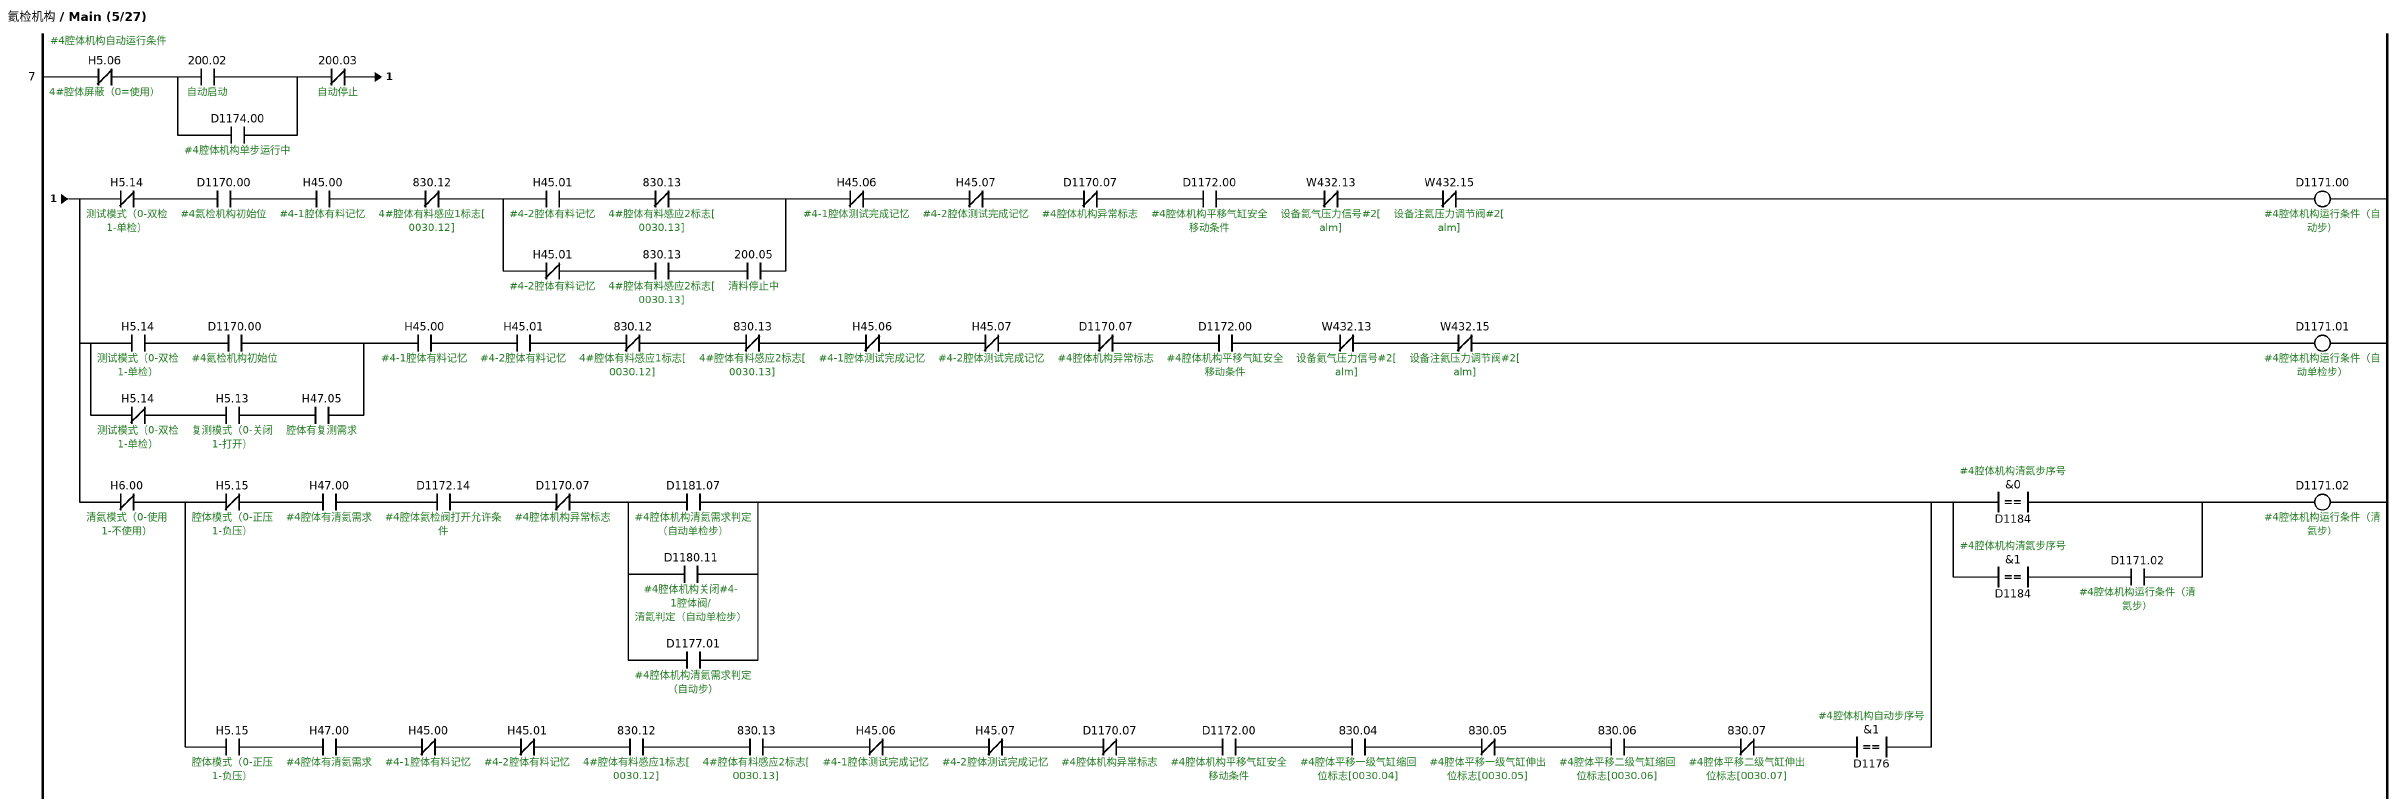
; [picture p144: 氦检机构 / Main, rungs 7-7]
; rung 7: #4腔体机构自动运行条件
LDNOT H5.06  ; 4#腔体屏蔽（0=使用）
LD 200.02  ; 自动启动
OR D1174.00  ; #4腔体机构单步运行中
ANDLD
ANDNOT 200.03  ; 自动停止
OUT TR0
ANDNOT H5.14  ; 测试模式（0-双检 1-单检）
AND D1170.00  ; #4氦检机构初始位
AND H45.00  ; #4-1腔体有料记忆
ANDNOT 830.12  ; 4#腔体有料感应1标志[0030.12]
LD H45.01  ; #4-2腔体有料记忆
ANDNOT 830.13  ; 4#腔体有料感应2标志[0030.13]
LDNOT H45.01  ; #4-2腔体有料记忆
AND 830.13  ; 4#腔体有料感应2标志[0030.13]
AND 200.05  ; 清料停止中
ORLD
ANDLD
ANDNOT H45.06  ; #4-1腔体测试完成记忆
ANDNOT H45.07  ; #4-2腔体测试完成记忆
ANDNOT D1170.07  ; #4腔体机构异常标志
AND D1172.00  ; #4腔体机构平移气缸安全移动条件
ANDNOT W432.13  ; 设备氦气压力信号#2[alm]
ANDNOT W432.15  ; 设备注氦压力调节阀#2[alm]
OUT D1171.00  ; #4腔体机构运行条件（自动步）
LD TR0
LD H5.14  ; 测试模式（0-双检 1-单检）
AND D1170.00  ; #4氦检机构初始位
LDNOT H5.14  ; 测试模式（0-双检 1-单检）
AND H5.13  ; 复测模式（0-关闭 1-打开）
AND H47.05  ; 腔体有复测需求
ORLD
ANDLD
AND H45.00  ; #4-1腔体有料记忆
AND H45.01  ; #4-2腔体有料记忆
ANDNOT 830.12  ; 4#腔体有料感应1标志[0030.12]
ANDNOT 830.13  ; 4#腔体有料感应2标志[0030.13]
ANDNOT H45.06  ; #4-1腔体测试完成记忆
ANDNOT H45.07  ; #4-2腔体测试完成记忆
ANDNOT D1170.07  ; #4腔体机构异常标志
AND D1172.00  ; #4腔体机构平移气缸安全移动条件
ANDNOT W432.13  ; 设备氦气压力信号#2[alm]
ANDNOT W432.15  ; 设备注氦压力调节阀#2[alm]
OUT D1171.01  ; #4腔体机构运行条件（自动单检步）
LD TR0
ANDNOT H6.00  ; 清氦模式（0-使用 1-不使用）
LDNOT H5.15  ; 腔体模式（0-正压 1-负压）
AND H47.00  ; #4腔体有清氦需求
AND D1172.14  ; #4腔体氦检阀打开允许条件
ANDNOT D1170.07  ; #4腔体机构异常标志
LD D1181.07  ; #4腔体机构清氦需求判定（自动单检步）
OR D1180.11  ; #4腔体机构关闭#4-1腔体阀/清氦判定（自动单检步）
OR D1177.01  ; #4腔体机构清氦需求判定（自动步）
ANDLD
LD H5.15  ; 腔体模式（0-正压 1-负压）
AND H47.00  ; #4腔体有清氦需求
ANDNOT H45.00  ; #4-1腔体有料记忆
ANDNOT H45.01  ; #4-2腔体有料记忆
AND 830.12  ; 4#腔体有料感应1标志[0030.12]
AND 830.13  ; 4#腔体有料感应2标志[0030.13]
ANDNOT H45.06  ; #4-1腔体测试完成记忆
ANDNOT H45.07  ; #4-2腔体测试完成记忆
ANDNOT D1170.07  ; #4腔体机构异常标志
AND D1172.00  ; #4腔体机构平移气缸安全移动条件
AND 830.04  ; #4腔体平移一级气缸缩回位标志[0030.04]
ANDNOT 830.05  ; #4腔体平移一级气缸伸出位标志[0030.05]
AND 830.06  ; #4腔体平移二级气缸缩回位标志[0030.06]
ANDNOT 830.07  ; #4腔体平移二级气缸伸出位标志[0030.07]
AND=L(301) &1 D1176  ; #4腔体机构自动步序号
ORLD
ANDLD
LD=L(301) &0 D1184  ; #4腔体机构清氦步序号
LD=L(301) &1 D1184  ; #4腔体机构清氦步序号
AND D1171.02  ; #4腔体机构运行条件（清氦步）
ORLD
ANDLD
OUT D1171.02  ; #4腔体机构运行条件（清氦步）

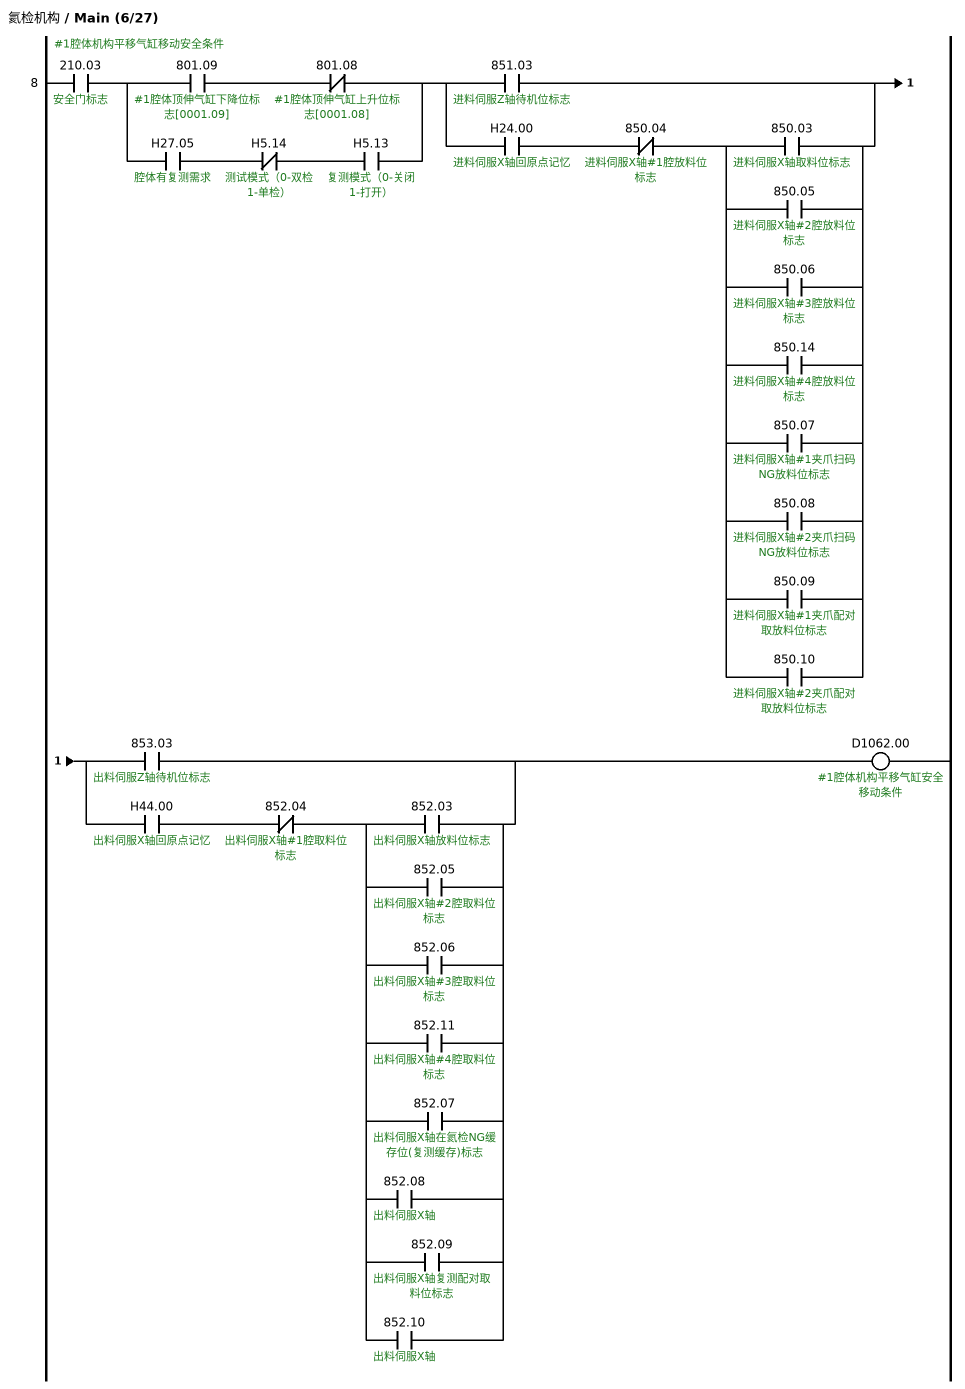
; rung 8: #1腔体机构平移气缸移动安全条件
LD 210.03  ; 安全门标志
LD 801.09  ; #1腔体顶伸气缸下降位标志[0001.09]
ANDNOT 801.08  ; #1腔体顶伸气缸上升位标志[0001.08]
LD H27.05  ; 腔体有复测需求
ANDNOT H5.14  ; 测试模式（0-双检 1-单检）
AND H5.13  ; 复测模式（0-关闭 1-打开）
ORLD
ANDLD
LD 851.03  ; 进料伺服Z轴待机位标志
LD H24.00  ; 进料伺服X轴回原点记忆
ANDNOT 850.04  ; 进料伺服X轴#1腔放料位标志
LD 850.03  ; 进料伺服X轴取料位标志
OR 850.05  ; 进料伺服X轴#2腔放料位标志
OR 850.06  ; 进料伺服X轴#3腔放料位标志
OR 850.14  ; 进料伺服X轴#4腔放料位标志
OR 850.07  ; 进料伺服X轴#1夹爪扫码NG放料位标志
OR 850.08  ; 进料伺服X轴#2夹爪扫码NG放料位标志
OR 850.09  ; 进料伺服X轴#1夹爪配对取放料位标志
OR 850.10  ; 进料伺服X轴#2夹爪配对取放料位标志
ANDLD
ORLD
ANDLD
LD 853.03  ; 出料伺服Z轴待机位标志
LD H44.00  ; 出料伺服X轴回原点记忆
ANDNOT 852.04  ; 出料伺服X轴#1腔取料位标志
LD 852.03  ; 出料伺服X轴放料位标志
OR 852.05  ; 出料伺服X轴#2腔取料位标志
OR 852.06  ; 出料伺服X轴#3腔取料位标志
OR 852.11  ; 出料伺服X轴#4腔取料位标志
OR 852.07  ; 出料伺服X轴在氦检NG缓存位(复测缓存)标志
OR 852.08  ; 出料伺服X轴
OR 852.09  ; 出料伺服X轴复测配对取料位标志
OR 852.10  ; 出料伺服X轴
ANDLD
ORLD
ANDLD
OUT D1062.00  ; #1腔体机构平移气缸安全移动条件

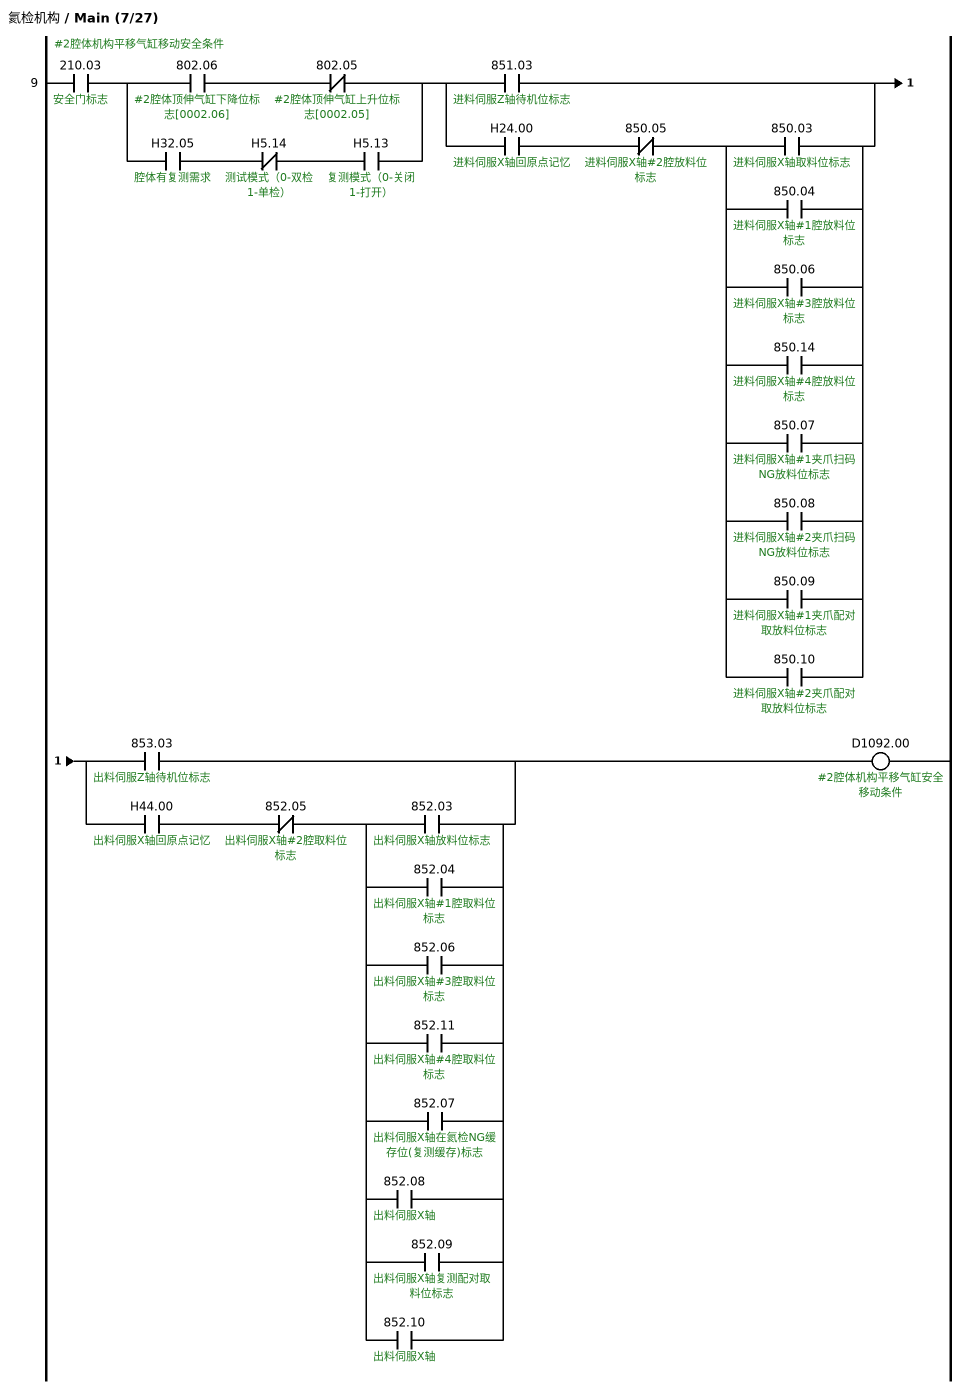
; rung 9: #2腔体机构平移气缸移动安全条件
LD 210.03  ; 安全门标志
LD 802.06  ; #2腔体顶伸气缸下降位标志[0002.06]
ANDNOT 802.05  ; #2腔体顶伸气缸上升位标志[0002.05]
LD H32.05  ; 腔体有复测需求
ANDNOT H5.14  ; 测试模式（0-双检 1-单检）
AND H5.13  ; 复测模式（0-关闭 1-打开）
ORLD
ANDLD
LD 851.03  ; 进料伺服Z轴待机位标志
LD H24.00  ; 进料伺服X轴回原点记忆
ANDNOT 850.05  ; 进料伺服X轴#2腔放料位标志
LD 850.03  ; 进料伺服X轴取料位标志
OR 850.04  ; 进料伺服X轴#1腔放料位标志
OR 850.06  ; 进料伺服X轴#3腔放料位标志
OR 850.14  ; 进料伺服X轴#4腔放料位标志
OR 850.07  ; 进料伺服X轴#1夹爪扫码NG放料位标志
OR 850.08  ; 进料伺服X轴#2夹爪扫码NG放料位标志
OR 850.09  ; 进料伺服X轴#1夹爪配对取放料位标志
OR 850.10  ; 进料伺服X轴#2夹爪配对取放料位标志
ANDLD
ORLD
ANDLD
LD 853.03  ; 出料伺服Z轴待机位标志
LD H44.00  ; 出料伺服X轴回原点记忆
ANDNOT 852.05  ; 出料伺服X轴#2腔取料位标志
LD 852.03  ; 出料伺服X轴放料位标志
OR 852.04  ; 出料伺服X轴#1腔取料位标志
OR 852.06  ; 出料伺服X轴#3腔取料位标志
OR 852.11  ; 出料伺服X轴#4腔取料位标志
OR 852.07  ; 出料伺服X轴在氦检NG缓存位(复测缓存)标志
OR 852.08  ; 出料伺服X轴
OR 852.09  ; 出料伺服X轴复测配对取料位标志
OR 852.10  ; 出料伺服X轴
ANDLD
ORLD
ANDLD
OUT D1092.00  ; #2腔体机构平移气缸安全移动条件

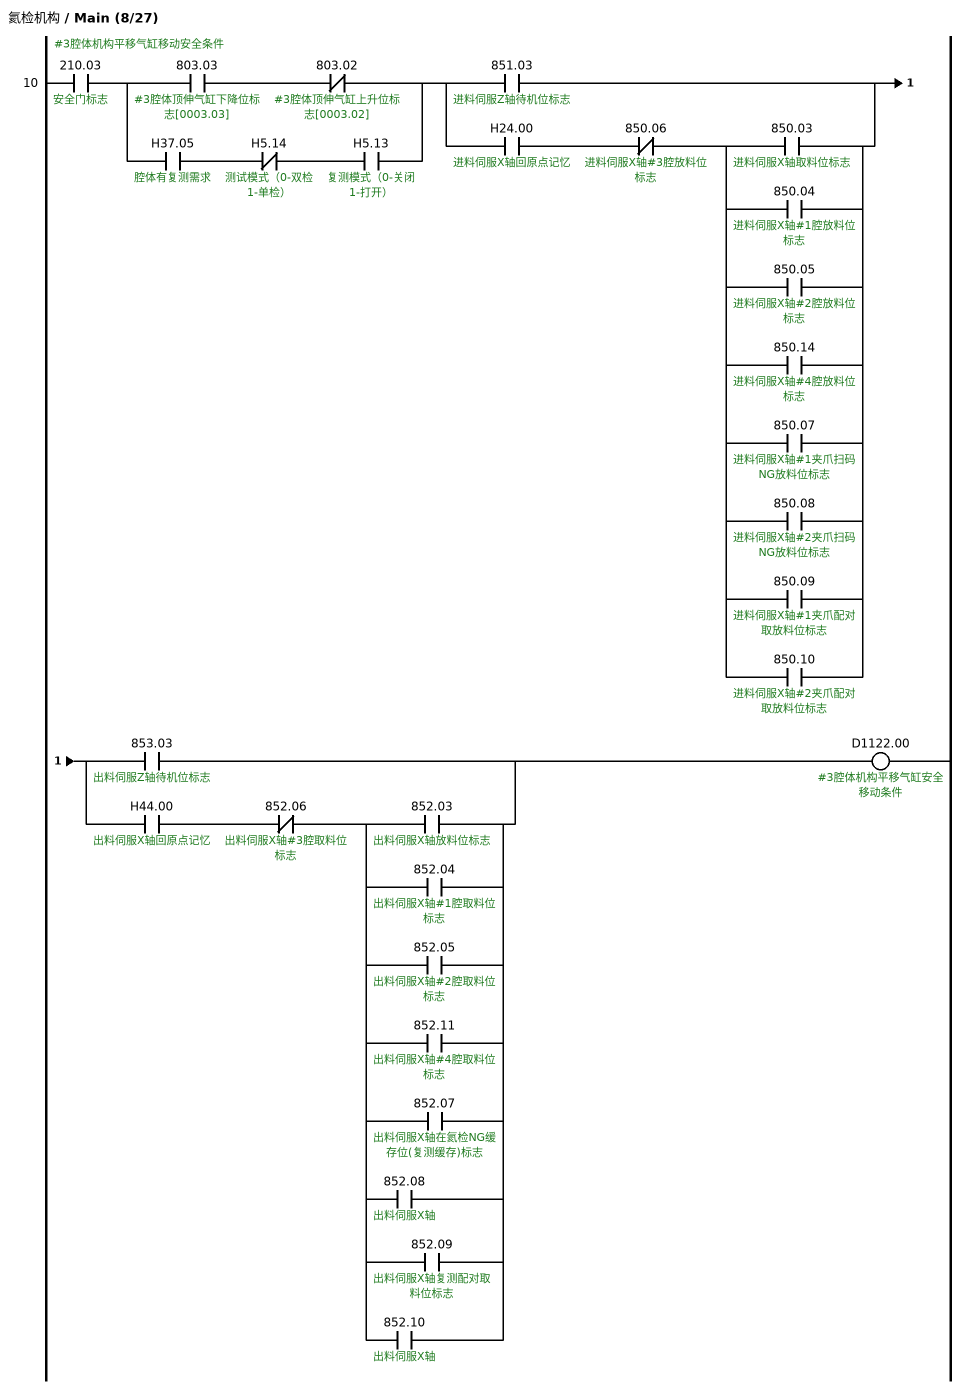
; rung 10: #3腔体机构平移气缸移动安全条件
LD 210.03  ; 安全门标志
LD 803.03  ; #3腔体顶伸气缸下降位标志[0003.03]
ANDNOT 803.02  ; #3腔体顶伸气缸上升位标志[0003.02]
LD H37.05  ; 腔体有复测需求
ANDNOT H5.14  ; 测试模式（0-双检 1-单检）
AND H5.13  ; 复测模式（0-关闭 1-打开）
ORLD
ANDLD
LD 851.03  ; 进料伺服Z轴待机位标志
LD H24.00  ; 进料伺服X轴回原点记忆
ANDNOT 850.06  ; 进料伺服X轴#3腔放料位标志
LD 850.03  ; 进料伺服X轴取料位标志
OR 850.04  ; 进料伺服X轴#1腔放料位标志
OR 850.05  ; 进料伺服X轴#2腔放料位标志
OR 850.14  ; 进料伺服X轴#4腔放料位标志
OR 850.07  ; 进料伺服X轴#1夹爪扫码NG放料位标志
OR 850.08  ; 进料伺服X轴#2夹爪扫码NG放料位标志
OR 850.09  ; 进料伺服X轴#1夹爪配对取放料位标志
OR 850.10  ; 进料伺服X轴#2夹爪配对取放料位标志
ANDLD
ORLD
ANDLD
LD 853.03  ; 出料伺服Z轴待机位标志
LD H44.00  ; 出料伺服X轴回原点记忆
ANDNOT 852.06  ; 出料伺服X轴#3腔取料位标志
LD 852.03  ; 出料伺服X轴放料位标志
OR 852.04  ; 出料伺服X轴#1腔取料位标志
OR 852.05  ; 出料伺服X轴#2腔取料位标志
OR 852.11  ; 出料伺服X轴#4腔取料位标志
OR 852.07  ; 出料伺服X轴在氦检NG缓存位(复测缓存)标志
OR 852.08  ; 出料伺服X轴
OR 852.09  ; 出料伺服X轴复测配对取料位标志
OR 852.10  ; 出料伺服X轴
ANDLD
ORLD
ANDLD
OUT D1122.00  ; #3腔体机构平移气缸安全移动条件

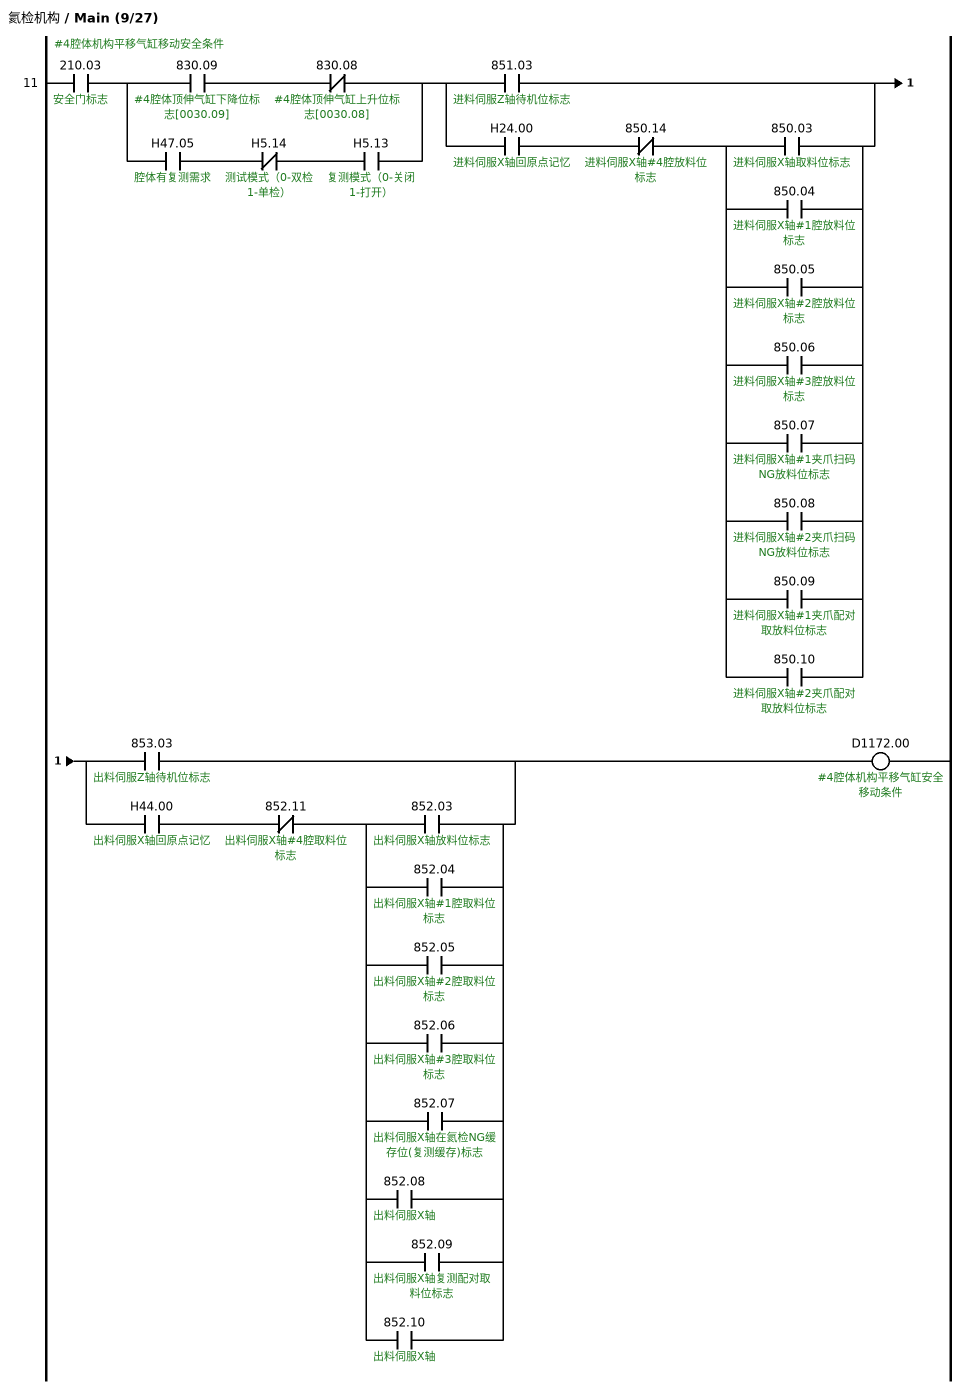
; rung 11: #4腔体机构平移气缸移动安全条件
LD 210.03  ; 安全门标志
LD 830.09  ; #4腔体顶伸气缸下降位标志[0030.09]
ANDNOT 830.08  ; #4腔体顶伸气缸上升位标志[0030.08]
LD H47.05  ; 腔体有复测需求
ANDNOT H5.14  ; 测试模式（0-双检 1-单检）
AND H5.13  ; 复测模式（0-关闭 1-打开）
ORLD
ANDLD
LD 851.03  ; 进料伺服Z轴待机位标志
LD H24.00  ; 进料伺服X轴回原点记忆
ANDNOT 850.14  ; 进料伺服X轴#4腔放料位标志
LD 850.03  ; 进料伺服X轴取料位标志
OR 850.04  ; 进料伺服X轴#1腔放料位标志
OR 850.05  ; 进料伺服X轴#2腔放料位标志
OR 850.06  ; 进料伺服X轴#3腔放料位标志
OR 850.07  ; 进料伺服X轴#1夹爪扫码NG放料位标志
OR 850.08  ; 进料伺服X轴#2夹爪扫码NG放料位标志
OR 850.09  ; 进料伺服X轴#1夹爪配对取放料位标志
OR 850.10  ; 进料伺服X轴#2夹爪配对取放料位标志
ANDLD
ORLD
ANDLD
LD 853.03  ; 出料伺服Z轴待机位标志
LD H44.00  ; 出料伺服X轴回原点记忆
ANDNOT 852.11  ; 出料伺服X轴#4腔取料位标志
LD 852.03  ; 出料伺服X轴放料位标志
OR 852.04  ; 出料伺服X轴#1腔取料位标志
OR 852.05  ; 出料伺服X轴#2腔取料位标志
OR 852.06  ; 出料伺服X轴#3腔取料位标志
OR 852.07  ; 出料伺服X轴在氦检NG缓存位(复测缓存)标志
OR 852.08  ; 出料伺服X轴
OR 852.09  ; 出料伺服X轴复测配对取料位标志
OR 852.10  ; 出料伺服X轴
ANDLD
ORLD
ANDLD
OUT D1172.00  ; #4腔体机构平移气缸安全移动条件

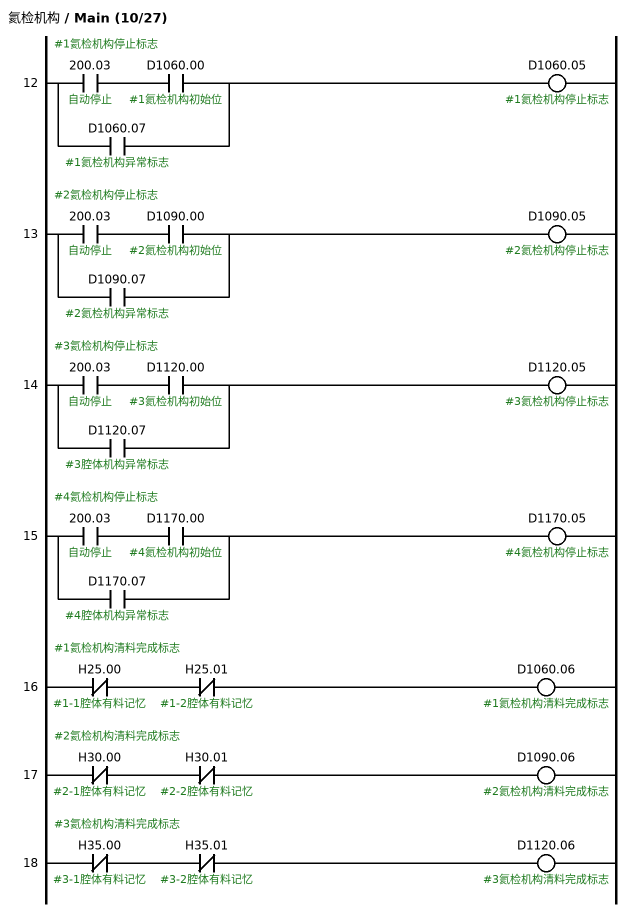
; rung 12: #1氦检机构停止标志
LD 200.03  ; 自动停止
AND D1060.00  ; #1氦检机构初始位
OR D1060.07  ; #1氦检机构异常标志
OUT D1060.05  ; #1氦检机构停止标志
; rung 13: #2氦检机构停止标志
LD 200.03  ; 自动停止
AND D1090.00  ; #2氦检机构初始位
OR D1090.07  ; #2氦检机构异常标志
OUT D1090.05  ; #2氦检机构停止标志
; rung 14: #3氦检机构停止标志
LD 200.03  ; 自动停止
AND D1120.00  ; #3氦检机构初始位
OR D1120.07  ; #3腔体机构异常标志
OUT D1120.05  ; #3氦检机构停止标志
; rung 15: #4氦检机构停止标志
LD 200.03  ; 自动停止
AND D1170.00  ; #4氦检机构初始位
OR D1170.07  ; #4腔体机构异常标志
OUT D1170.05  ; #4氦检机构停止标志
; rung 16: #1氦检机构清料完成标志
LDNOT H25.00  ; #1-1腔体有料记忆
ANDNOT H25.01  ; #1-2腔体有料记忆
OUT D1060.06  ; #1氦检机构清料完成标志
; rung 17: #2氦检机构清料完成标志
LDNOT H30.00  ; #2-1腔体有料记忆
ANDNOT H30.01  ; #2-2腔体有料记忆
OUT D1090.06  ; #2氦检机构清料完成标志
; rung 18: #3氦检机构清料完成标志
LDNOT H35.00  ; #3-1腔体有料记忆
ANDNOT H35.01  ; #3-2腔体有料记忆
OUT D1120.06  ; #3氦检机构清料完成标志

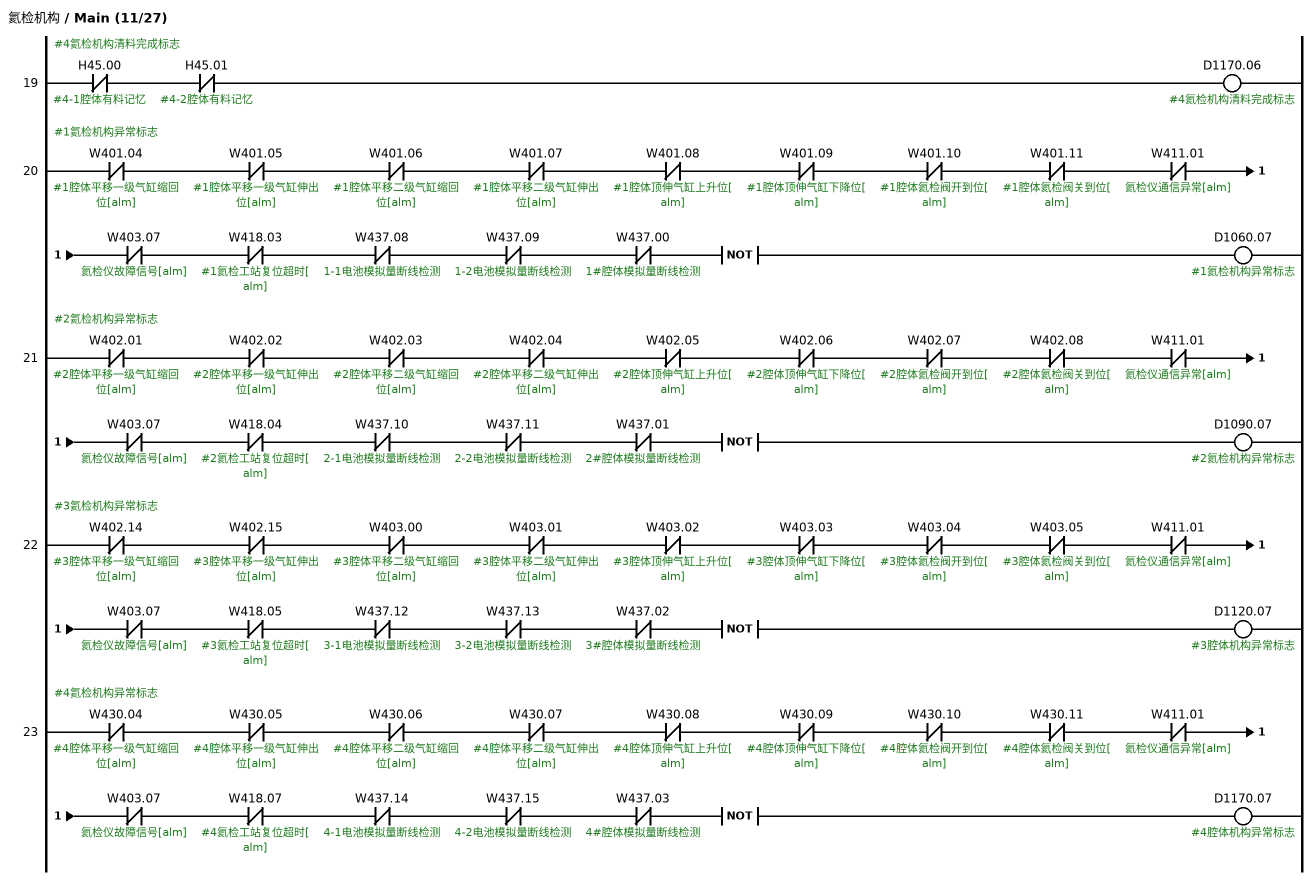
; rung 19: #4氦检机构清料完成标志
LDNOT H45.00  ; #4-1腔体有料记忆
ANDNOT H45.01  ; #4-2腔体有料记忆
OUT D1170.06  ; #4氦检机构清料完成标志
; rung 20: #1氦检机构异常标志
LDNOT W401.04  ; #1腔体平移一级气缸缩回位[alm]
ANDNOT W401.05  ; #1腔体平移一级气缸伸出位[alm]
ANDNOT W401.06  ; #1腔体平移二级气缸缩回位[alm]
ANDNOT W401.07  ; #1腔体平移二级气缸伸出位[alm]
ANDNOT W401.08  ; #1腔体顶伸气缸上升位[alm]
ANDNOT W401.09  ; #1腔体顶伸气缸下降位[alm]
ANDNOT W401.10  ; #1腔体氦检阀开到位[alm]
ANDNOT W401.11  ; #1腔体氦检阀关到位[alm]
ANDNOT W411.01  ; 氦检仪通信异常[alm]
ANDNOT W403.07  ; 氦检仪故障信号[alm]
ANDNOT W418.03  ; #1氦检工站复位超时[alm]
ANDNOT W437.08  ; 1-1电池模拟量断线检测
ANDNOT W437.09  ; 1-2电池模拟量断线检测
ANDNOT W437.00  ; 1#腔体模拟量断线检测
NOT(520)
OUT D1060.07  ; #1氦检机构异常标志
; rung 21: #2氦检机构异常标志
LDNOT W402.01  ; #2腔体平移一级气缸缩回位[alm]
ANDNOT W402.02  ; #2腔体平移一级气缸伸出位[alm]
ANDNOT W402.03  ; #2腔体平移二级气缸缩回位[alm]
ANDNOT W402.04  ; #2腔体平移二级气缸伸出位[alm]
ANDNOT W402.05  ; #2腔体顶伸气缸上升位[alm]
ANDNOT W402.06  ; #2腔体顶伸气缸下降位[alm]
ANDNOT W402.07  ; #2腔体氦检阀开到位[alm]
ANDNOT W402.08  ; #2腔体氦检阀关到位[alm]
ANDNOT W411.01  ; 氦检仪通信异常[alm]
ANDNOT W403.07  ; 氦检仪故障信号[alm]
ANDNOT W418.04  ; #2氦检工站复位超时[alm]
ANDNOT W437.10  ; 2-1电池模拟量断线检测
ANDNOT W437.11  ; 2-2电池模拟量断线检测
ANDNOT W437.01  ; 2#腔体模拟量断线检测
NOT(520)
OUT D1090.07  ; #2氦检机构异常标志
; rung 22: #3氦检机构异常标志
LDNOT W402.14  ; #3腔体平移一级气缸缩回位[alm]
ANDNOT W402.15  ; #3腔体平移一级气缸伸出位[alm]
ANDNOT W403.00  ; #3腔体平移二级气缸缩回位[alm]
ANDNOT W403.01  ; #3腔体平移二级气缸伸出位[alm]
ANDNOT W403.02  ; #3腔体顶伸气缸上升位[alm]
ANDNOT W403.03  ; #3腔体顶伸气缸下降位[alm]
ANDNOT W403.04  ; #3腔体氦检阀开到位[alm]
ANDNOT W403.05  ; #3腔体氦检阀关到位[alm]
ANDNOT W411.01  ; 氦检仪通信异常[alm]
ANDNOT W403.07  ; 氦检仪故障信号[alm]
ANDNOT W418.05  ; #3氦检工站复位超时[alm]
ANDNOT W437.12  ; 3-1电池模拟量断线检测
ANDNOT W437.13  ; 3-2电池模拟量断线检测
ANDNOT W437.02  ; 3#腔体模拟量断线检测
NOT(520)
OUT D1120.07  ; #3腔体机构异常标志
; rung 23: #4氦检机构异常标志
LDNOT W430.04  ; #4腔体平移一级气缸缩回位[alm]
ANDNOT W430.05  ; #4腔体平移一级气缸伸出位[alm]
ANDNOT W430.06  ; #4腔体平移二级气缸缩回位[alm]
ANDNOT W430.07  ; #4腔体平移二级气缸伸出位[alm]
ANDNOT W430.08  ; #4腔体顶伸气缸上升位[alm]
ANDNOT W430.09  ; #4腔体顶伸气缸下降位[alm]
ANDNOT W430.10  ; #4腔体氦检阀开到位[alm]
ANDNOT W430.11  ; #4腔体氦检阀关到位[alm]
ANDNOT W411.01  ; 氦检仪通信异常[alm]
ANDNOT W403.07  ; 氦检仪故障信号[alm]
ANDNOT W418.07  ; #4氦检工站复位超时[alm]
ANDNOT W437.14  ; 4-1电池模拟量断线检测
ANDNOT W437.15  ; 4-2电池模拟量断线检测
ANDNOT W437.03  ; 4#腔体模拟量断线检测
NOT(520)
OUT D1170.07  ; #4腔体机构异常标志

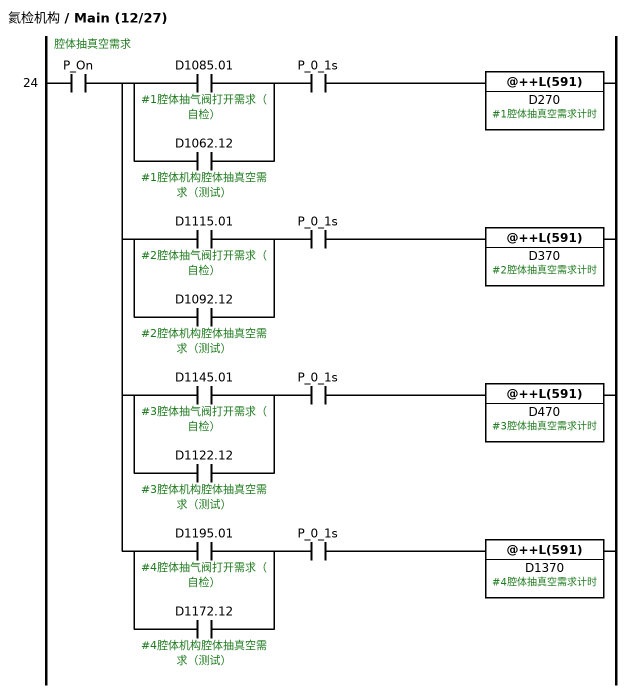
; rung 24: 腔体抽真空需求
LD P_On
OUT TR0
LD D1085.01  ; #1腔体抽气阀打开需求（自检）
OR D1062.12  ; #1腔体机构腔体抽真空需求（测试）
ANDLD
AND P_0_1s
@++L(591) D270  ; #1腔体抽真空需求计时
LD TR0
LD D1115.01  ; #2腔体抽气阀打开需求（自检）
OR D1092.12  ; #2腔体机构腔体抽真空需求（测试）
ANDLD
AND P_0_1s
@++L(591) D370  ; #2腔体抽真空需求计时
LD TR0
LD D1145.01  ; #3腔体抽气阀打开需求（自检）
OR D1122.12  ; #3腔体机构腔体抽真空需求（测试）
ANDLD
AND P_0_1s
@++L(591) D470  ; #3腔体抽真空需求计时
LD TR0
LD D1195.01  ; #4腔体抽气阀打开需求（自检）
OR D1172.12  ; #4腔体机构腔体抽真空需求（测试）
ANDLD
AND P_0_1s
@++L(591) D1370  ; #4腔体抽真空需求计时

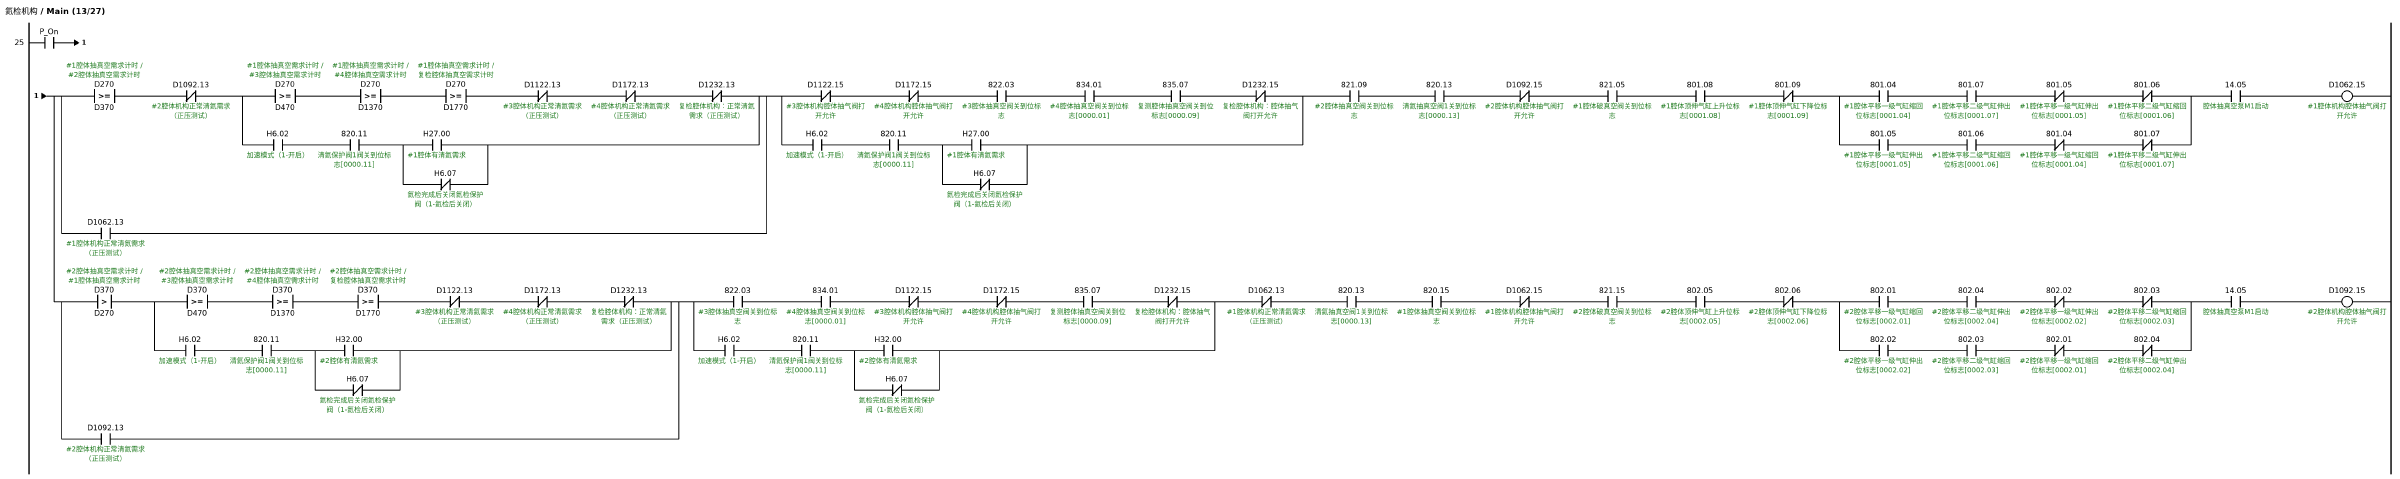
; rung 25
LD P_On
OUT TR0
LD>=L(326) D270 D370  ; #1腔体抽真空需求计时, #2腔体抽真空需求计时
ANDNOT D1092.13  ; #2腔体机构正常清氦需求（正压测试）
LD>=L(326) D270 D470  ; #1腔体抽真空需求计时, #3腔体抽真空需求计时
AND>=L(326) D270 D1370  ; #1腔体抽真空需求计时, #4腔体抽真空需求计时
AND>=L(326) D270 D1770  ; #1腔体抽真空需求计时, 复检腔体抽真空需求计时
ANDNOT D1122.13  ; #3腔体机构正常清氦需求（正压测试）
ANDNOT D1172.13  ; #4腔体机构正常清氦需求（正压测试）
ANDNOT D1232.13  ; 复检腔体机构：正常清氦需求（正压测试）
LD H6.02  ; 加速模式（1-开启）
AND 820.11  ; 清氦保护阀1阀关到位标志[0000.11]
LD H27.00  ; #1腔体有清氦需求
ORNOT H6.07  ; 氦检完成后关闭氦检保护阀（1-氦检后关闭）
ANDLD
ORLD
ANDLD
OR D1062.13  ; #1腔体机构正常清氦需求（正压测试）
ANDLD
LDNOT D1122.15  ; #3腔体机构腔体抽气阀打开允许
ANDNOT D1172.15  ; #4腔体机构腔体抽气阀打开允许
AND 822.03  ; #3腔体抽真空阀关到位标志
AND 834.01  ; #4腔体抽真空阀关到位标志[0000.01]
AND 835.07  ; 复测腔体抽真空阀关到位标志[0000.09]
ANDNOT D1232.15  ; 复检腔体机构：腔体抽气阀打开允许
LD H6.02  ; 加速模式（1-开启）
AND 820.11  ; 清氦保护阀1阀关到位标志[0000.11]
LD H27.00  ; #1腔体有清氦需求
ORNOT H6.07  ; 氦检完成后关闭氦检保护阀（1-氦检后关闭）
ANDLD
ORLD
ANDLD
AND 821.09  ; #2腔体抽真空阀关到位标志
AND 820.13  ; 清氦抽真空阀1关到位标志[0000.13]
ANDNOT D1092.15  ; #2腔体机构腔体抽气阀打开允许
AND 821.05  ; #1腔体破真空阀关到位标志
AND 801.08  ; #1腔体顶伸气缸上升位标志[0001.08]
ANDNOT 801.09  ; #1腔体顶伸气缸下降位标志[0001.09]
LD 801.04  ; #1腔体平移一级气缸缩回位标志[0001.04]
AND 801.07  ; #1腔体平移二级气缸伸出位标志[0001.07]
ANDNOT 801.05  ; #1腔体平移一级气缸伸出位标志[0001.05]
ANDNOT 801.06  ; #1腔体平移二级气缸缩回位标志[0001.06]
LD 801.05  ; #1腔体平移一级气缸伸出位标志[0001.05]
AND 801.06  ; #1腔体平移二级气缸缩回位标志[0001.06]
ANDNOT 801.04  ; #1腔体平移一级气缸缩回位标志[0001.04]
ANDNOT 801.07  ; #1腔体平移二级气缸伸出位标志[0001.07]
ORLD
ANDLD
AND 14.05  ; 腔体抽真空泵M1启动
OUT D1062.15  ; #1腔体机构腔体抽气阀打开允许
LD TR0
LD>L(321) D370 D270  ; #2腔体抽真空需求计时, #1腔体抽真空需求计时
LD>=L(326) D370 D470  ; #2腔体抽真空需求计时, #3腔体抽真空需求计时
AND>=L(326) D370 D1370  ; #2腔体抽真空需求计时, #4腔体抽真空需求计时
AND>=L(326) D370 D1770  ; #2腔体抽真空需求计时, 复检腔体抽真空需求计时
ANDNOT D1122.13  ; #3腔体机构正常清氦需求（正压测试）
ANDNOT D1172.13  ; #4腔体机构正常清氦需求（正压测试）
ANDNOT D1232.13  ; 复检腔体机构：正常清氦需求（正压测试）
LD H6.02  ; 加速模式（1-开启）
AND 820.11  ; 清氦保护阀1阀关到位标志[0000.11]
LD H32.00  ; #2腔体有清氦需求
ORNOT H6.07  ; 氦检完成后关闭氦检保护阀（1-氦检后关闭）
ANDLD
ORLD
ANDLD
OR D1092.13  ; #2腔体机构正常清氦需求（正压测试）
ANDLD
LD 822.03  ; #3腔体抽真空阀关到位标志
AND 834.01  ; #4腔体抽真空阀关到位标志[0000.01]
ANDNOT D1122.15  ; #3腔体机构腔体抽气阀打开允许
ANDNOT D1172.15  ; #4腔体机构腔体抽气阀打开允许
AND 835.07  ; 复测腔体抽真空阀关到位标志[0000.09]
ANDNOT D1232.15  ; 复检腔体机构：腔体抽气阀打开允许
LD H6.02  ; 加速模式（1-开启）
AND 820.11  ; 清氦保护阀1阀关到位标志[0000.11]
LD H32.00  ; #2腔体有清氦需求
ORNOT H6.07  ; 氦检完成后关闭氦检保护阀（1-氦检后关闭）
ANDLD
ORLD
ANDLD
ANDNOT D1062.13  ; #1腔体机构正常清氦需求（正压测试）
AND 820.13  ; 清氦抽真空阀1关到位标志[0000.13]
AND 820.15  ; #1腔体抽真空阀关到位标志
ANDNOT D1062.15  ; #1腔体机构腔体抽气阀打开允许
AND 821.15  ; #2腔体破真空阀关到位标志
AND 802.05  ; #2腔体顶伸气缸上升位标志[0002.05]
ANDNOT 802.06  ; #2腔体顶伸气缸下降位标志[0002.06]
LD 802.01  ; #2腔体平移一级气缸缩回位标志[0002.01]
AND 802.04  ; #2腔体平移二级气缸伸出位标志[0002.04]
ANDNOT 802.02  ; #2腔体平移一级气缸伸出位标志[0002.02]
ANDNOT 802.03  ; #2腔体平移二级气缸缩回位标志[0002.03]
LD 802.02  ; #2腔体平移一级气缸伸出位标志[0002.02]
AND 802.03  ; #2腔体平移二级气缸缩回位标志[0002.03]
ANDNOT 802.01  ; #2腔体平移一级气缸缩回位标志[0002.01]
ANDNOT 802.04  ; #2腔体平移二级气缸伸出位标志[0002.04]
ORLD
ANDLD
AND 14.05  ; 腔体抽真空泵M1启动
OUT D1092.15  ; #2腔体机构腔体抽气阀打开允许

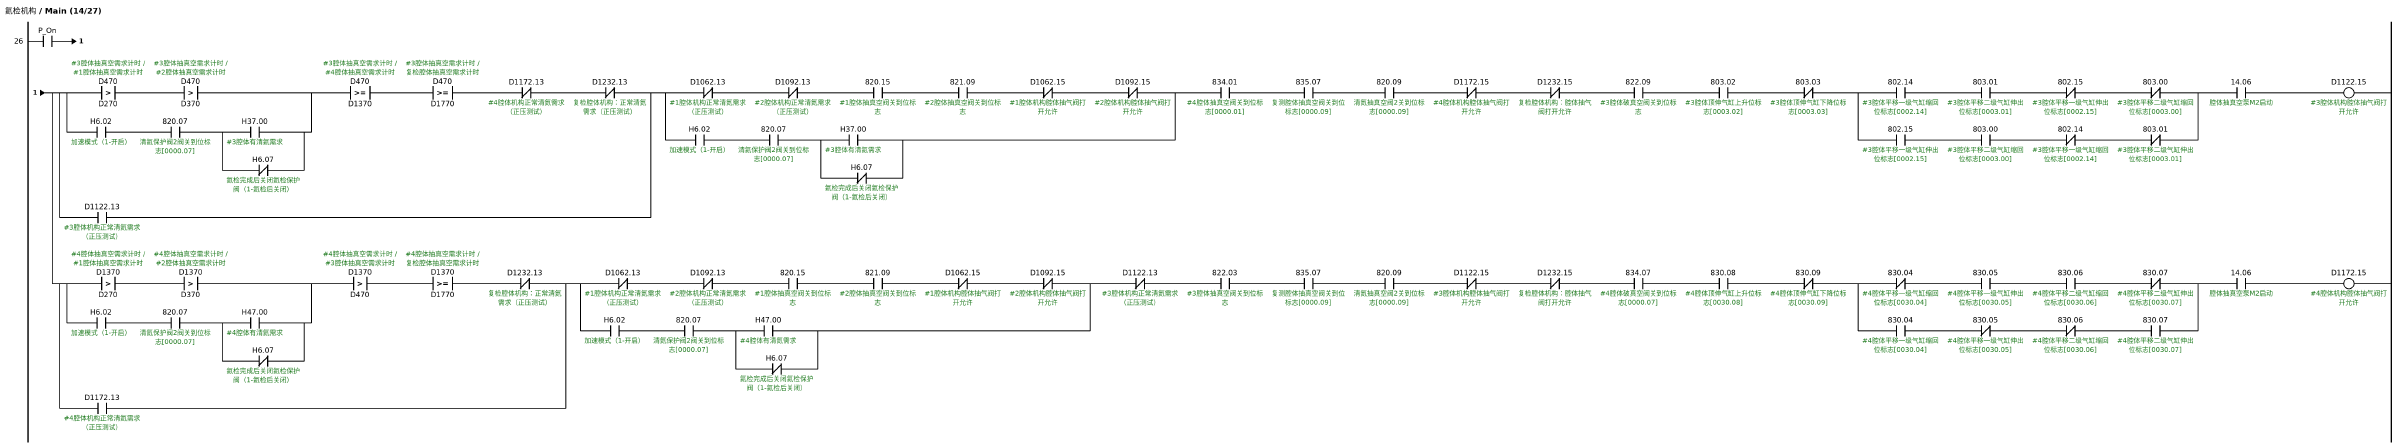
; rung 26
LD P_On
OUT TR0
LD>L(321) D470 D270  ; #3腔体抽真空需求计时, #1腔体抽真空需求计时
AND>L(321) D470 D370  ; #3腔体抽真空需求计时, #2腔体抽真空需求计时
LD H6.02  ; 加速模式（1-开启）
AND 820.07  ; 清氦保护阀2阀关到位标志[0000.07]
LD H37.00  ; #3腔体有清氦需求
ORNOT H6.07  ; 氦检完成后关闭氦检保护阀（1-氦检后关闭）
ANDLD
ORLD
AND>=L(326) D470 D1370  ; #3腔体抽真空需求计时, #4腔体抽真空需求计时
AND>=L(326) D470 D1770  ; #3腔体抽真空需求计时, 复检腔体抽真空需求计时
ANDNOT D1172.13  ; #4腔体机构正常清氦需求（正压测试）
ANDNOT D1232.13  ; 复检腔体机构：正常清氦需求（正压测试）
OR D1122.13  ; #3腔体机构正常清氦需求（正压测试）
ANDLD
LDNOT D1062.13  ; #1腔体机构正常清氦需求（正压测试）
ANDNOT D1092.13  ; #2腔体机构正常清氦需求（正压测试）
AND 820.15  ; #1腔体抽真空阀关到位标志
AND 821.09  ; #2腔体抽真空阀关到位标志
ANDNOT D1062.15  ; #1腔体机构腔体抽气阀打开允许
ANDNOT D1092.15  ; #2腔体机构腔体抽气阀打开允许
LD H6.02  ; 加速模式（1-开启）
AND 820.07  ; 清氦保护阀2阀关到位标志[0000.07]
LD H37.00  ; #3腔体有清氦需求
ORNOT H6.07  ; 氦检完成后关闭氦检保护阀（1-氦检后关闭）
ANDLD
ORLD
ANDLD
AND 834.01  ; #4腔体抽真空阀关到位标志[0000.01]
AND 835.07  ; 复测腔体抽真空阀关到位标志[0000.09]
AND 820.09  ; 清氦抽真空阀2关到位标志[0000.09]
ANDNOT D1172.15  ; #4腔体机构腔体抽气阀打开允许
ANDNOT D1232.15  ; 复检腔体机构：腔体抽气阀打开允许
AND 822.09  ; #3腔体破真空阀关到位标志
AND 803.02  ; #3腔体顶伸气缸上升位标志[0003.02]
ANDNOT 803.03  ; #3腔体顶伸气缸下降位标志[0003.03]
LD 802.14  ; #3腔体平移一级气缸缩回位标志[0002.14]
AND 803.01  ; #3腔体平移二级气缸伸出位标志[0003.01]
ANDNOT 802.15  ; #3腔体平移一级气缸伸出位标志[0002.15]
ANDNOT 803.00  ; #3腔体平移二级气缸缩回位标志[0003.00]
LD 802.15  ; #3腔体平移一级气缸伸出位标志[0002.15]
AND 803.00  ; #3腔体平移二级气缸缩回位标志[0003.00]
ANDNOT 802.14  ; #3腔体平移一级气缸缩回位标志[0002.14]
ANDNOT 803.01  ; #3腔体平移二级气缸伸出位标志[0003.01]
ORLD
ANDLD
AND 14.06  ; 腔体抽真空泵M2启动
OUT D1122.15  ; #3腔体机构腔体抽气阀打开允许
LD TR0
LD>L(321) D1370 D270  ; #4腔体抽真空需求计时, #1腔体抽真空需求计时
AND>L(321) D1370 D370  ; #4腔体抽真空需求计时, #2腔体抽真空需求计时
LD H6.02  ; 加速模式（1-开启）
AND 820.07  ; 清氦保护阀2阀关到位标志[0000.07]
LD H47.00  ; #4腔体有清氦需求
ORNOT H6.07  ; 氦检完成后关闭氦检保护阀（1-氦检后关闭）
ANDLD
ORLD
AND>L(321) D1370 D470  ; #4腔体抽真空需求计时, #3腔体抽真空需求计时
AND>=L(326) D1370 D1770  ; #4腔体抽真空需求计时, 复检腔体抽真空需求计时
ANDNOT D1232.13  ; 复检腔体机构：正常清氦需求（正压测试）
OR D1172.13  ; #4腔体机构正常清氦需求（正压测试）
ANDLD
LDNOT D1062.13  ; #1腔体机构正常清氦需求（正压测试）
ANDNOT D1092.13  ; #2腔体机构正常清氦需求（正压测试）
AND 820.15  ; #1腔体抽真空阀关到位标志
AND 821.09  ; #2腔体抽真空阀关到位标志
ANDNOT D1062.15  ; #1腔体机构腔体抽气阀打开允许
ANDNOT D1092.15  ; #2腔体机构腔体抽气阀打开允许
LD H6.02  ; 加速模式（1-开启）
AND 820.07  ; 清氦保护阀2阀关到位标志[0000.07]
LD H47.00  ; #4腔体有清氦需求
ORNOT H6.07  ; 氦检完成后关闭氦检保护阀（1-氦检后关闭）
ANDLD
ORLD
ANDLD
ANDNOT D1122.13  ; #3腔体机构正常清氦需求（正压测试）
AND 822.03  ; #3腔体抽真空阀关到位标志
AND 835.07  ; 复测腔体抽真空阀关到位标志[0000.09]
AND 820.09  ; 清氦抽真空阀2关到位标志[0000.09]
ANDNOT D1122.15  ; #3腔体机构腔体抽气阀打开允许
ANDNOT D1232.15  ; 复检腔体机构：腔体抽气阀打开允许
AND 834.07  ; #4腔体破真空阀关到位标志[0000.07]
AND 830.08  ; #4腔体顶伸气缸上升位标志[0030.08]
ANDNOT 830.09  ; #4腔体顶伸气缸下降位标志[0030.09]
LDNOT 830.04  ; #4腔体平移一级气缸缩回位标志[0030.04]
AND 830.05  ; #4腔体平移一级气缸伸出位标志[0030.05]
AND 830.06  ; #4腔体平移二级气缸缩回位标志[0030.06]
ANDNOT 830.07  ; #4腔体平移二级气缸伸出位标志[0030.07]
LD 830.04  ; #4腔体平移一级气缸缩回位标志[0030.04]
ANDNOT 830.05  ; #4腔体平移一级气缸伸出位标志[0030.05]
ANDNOT 830.06  ; #4腔体平移二级气缸缩回位标志[0030.06]
AND 830.07  ; #4腔体平移二级气缸伸出位标志[0030.07]
ORLD
ANDLD
AND 14.06  ; 腔体抽真空泵M2启动
OUT D1172.15  ; #4腔体机构腔体抽气阀打开允许

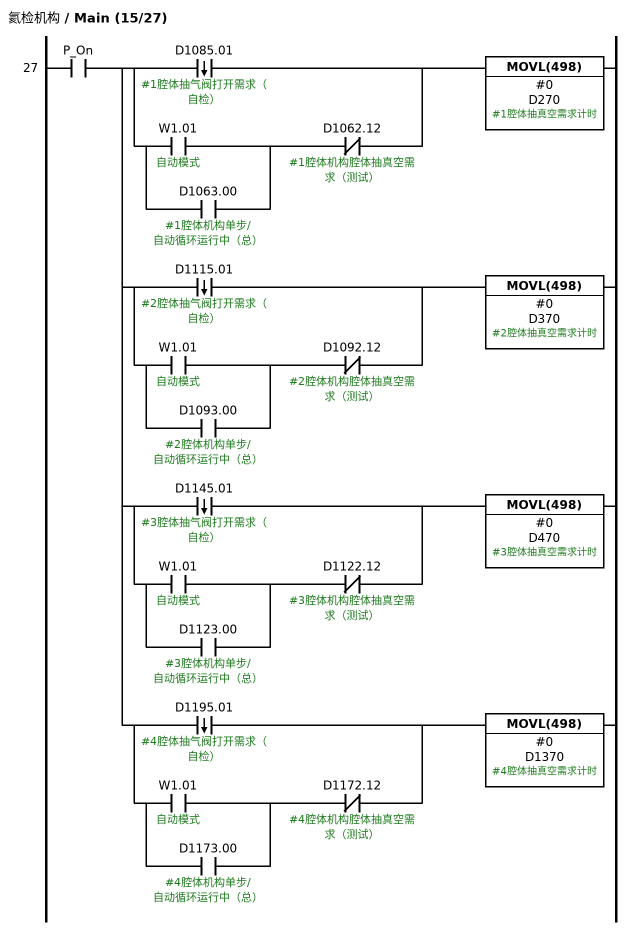
; rung 27
LD P_On
OUT TR0
%LD D1085.01  ; #1腔体抽气阀打开需求（自检）
LD W1.01  ; 自动模式
OR D1063.00  ; #1腔体机构单步/自动循环运行中（总）
ANDNOT D1062.12  ; #1腔体机构腔体抽真空需求（测试）
ORLD
ANDLD
MOVL(498) #0 D270  ; #1腔体抽真空需求计时
LD TR0
%LD D1115.01  ; #2腔体抽气阀打开需求（自检）
LD W1.01  ; 自动模式
OR D1093.00  ; #2腔体机构单步/自动循环运行中（总）
ANDNOT D1092.12  ; #2腔体机构腔体抽真空需求（测试）
ORLD
ANDLD
MOVL(498) #0 D370  ; #2腔体抽真空需求计时
LD TR0
%LD D1145.01  ; #3腔体抽气阀打开需求（自检）
LD W1.01  ; 自动模式
OR D1123.00  ; #3腔体机构单步/自动循环运行中（总）
ANDNOT D1122.12  ; #3腔体机构腔体抽真空需求（测试）
ORLD
ANDLD
MOVL(498) #0 D470  ; #3腔体抽真空需求计时
LD TR0
%LD D1195.01  ; #4腔体抽气阀打开需求（自检）
LD W1.01  ; 自动模式
OR D1173.00  ; #4腔体机构单步/自动循环运行中（总）
ANDNOT D1172.12  ; #4腔体机构腔体抽真空需求（测试）
ORLD
ANDLD
MOVL(498) #0 D1370  ; #4腔体抽真空需求计时

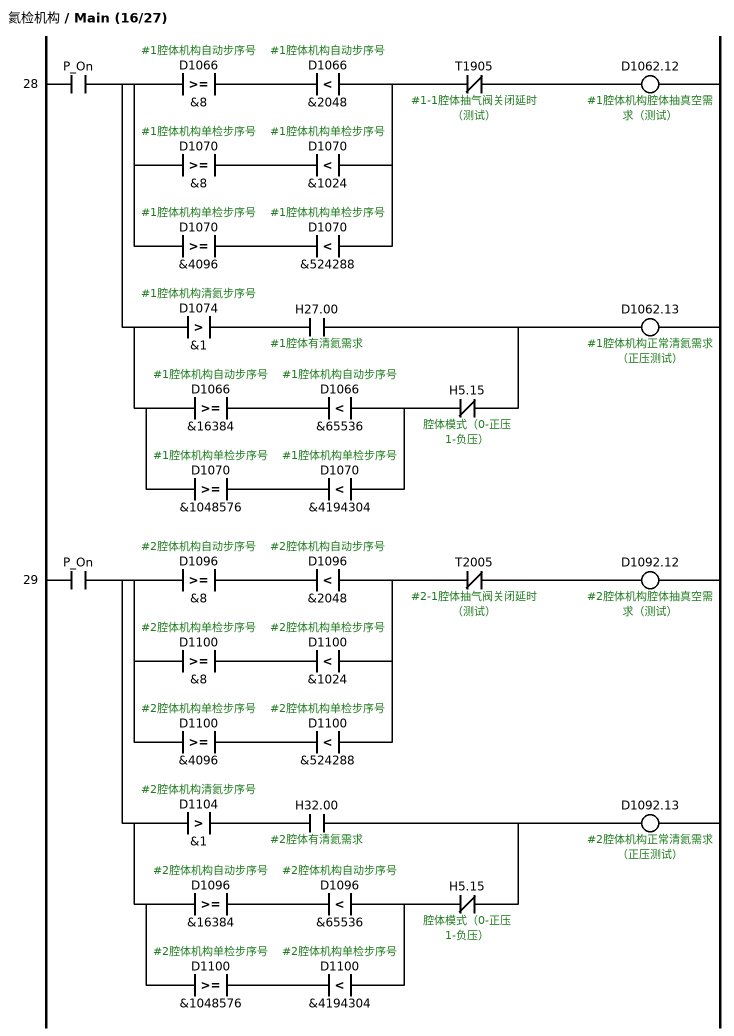
; rung 28
LD P_On
OUT TR0
LD>=L(326) D1066 &8  ; #1腔体机构自动步序号
AND<L(311) D1066 &2048  ; #1腔体机构自动步序号
LD>=L(326) D1070 &8  ; #1腔体机构单检步序号
AND<L(311) D1070 &1024  ; #1腔体机构单检步序号
ORLD
LD>=L(326) D1070 &4096  ; #1腔体机构单检步序号
AND<L(311) D1070 &524288  ; #1腔体机构单检步序号
ORLD
ANDLD
ANDNOT T1905  ; #1-1腔体抽气阀关闭延时（测试）
OUT D1062.12  ; #1腔体机构腔体抽真空需求（测试）
LD TR0
LD>L(321) D1074 &1  ; #1腔体机构清氦步序号
AND H27.00  ; #1腔体有清氦需求
LD>=L(326) D1066 &16384  ; #1腔体机构自动步序号
AND<L(311) D1066 &65536  ; #1腔体机构自动步序号
LD>=L(326) D1070 &1048576  ; #1腔体机构单检步序号
AND<L(311) D1070 &4194304  ; #1腔体机构单检步序号
ORLD
ANDNOT H5.15  ; 腔体模式（0-正压 1-负压）
ORLD
ANDLD
OUT D1062.13  ; #1腔体机构正常清氦需求（正压测试）
; rung 29
LD P_On
OUT TR0
LD>=L(326) D1096 &8  ; #2腔体机构自动步序号
AND<L(311) D1096 &2048  ; #2腔体机构自动步序号
LD>=L(326) D1100 &8  ; #2腔体机构单检步序号
AND<L(311) D1100 &1024  ; #2腔体机构单检步序号
ORLD
LD>=L(326) D1100 &4096  ; #2腔体机构单检步序号
AND<L(311) D1100 &524288  ; #2腔体机构单检步序号
ORLD
ANDLD
ANDNOT T2005  ; #2-1腔体抽气阀关闭延时（测试）
OUT D1092.12  ; #2腔体机构腔体抽真空需求（测试）
LD TR0
LD>L(321) D1104 &1  ; #2腔体机构清氦步序号
AND H32.00  ; #2腔体有清氦需求
LD>=L(326) D1096 &16384  ; #2腔体机构自动步序号
AND<L(311) D1096 &65536  ; #2腔体机构自动步序号
LD>=L(326) D1100 &1048576  ; #2腔体机构单检步序号
AND<L(311) D1100 &4194304  ; #2腔体机构单检步序号
ORLD
ANDNOT H5.15  ; 腔体模式（0-正压 1-负压）
ORLD
ANDLD
OUT D1092.13  ; #2腔体机构正常清氦需求（正压测试）

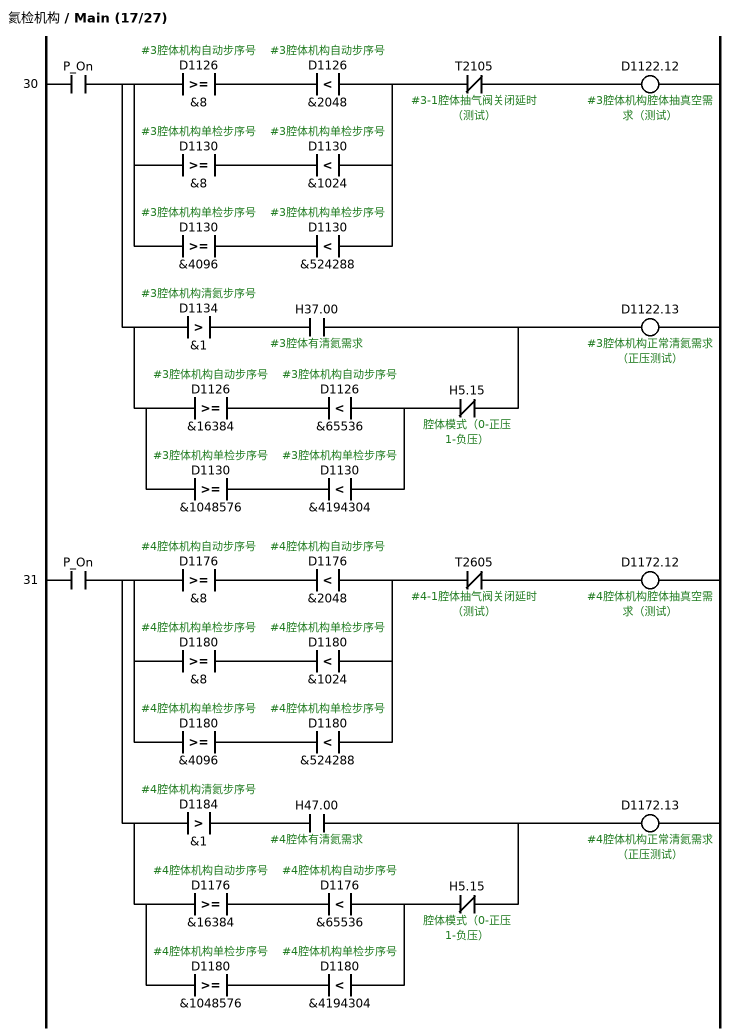
; rung 30
LD P_On
OUT TR0
LD>=L(326) D1126 &8  ; #3腔体机构自动步序号
AND<L(311) D1126 &2048  ; #3腔体机构自动步序号
LD>=L(326) D1130 &8  ; #3腔体机构单检步序号
AND<L(311) D1130 &1024  ; #3腔体机构单检步序号
ORLD
LD>=L(326) D1130 &4096  ; #3腔体机构单检步序号
AND<L(311) D1130 &524288  ; #3腔体机构单检步序号
ORLD
ANDLD
ANDNOT T2105  ; #3-1腔体抽气阀关闭延时（测试）
OUT D1122.12  ; #3腔体机构腔体抽真空需求（测试）
LD TR0
LD>L(321) D1134 &1  ; #3腔体机构清氦步序号
AND H37.00  ; #3腔体有清氦需求
LD>=L(326) D1126 &16384  ; #3腔体机构自动步序号
AND<L(311) D1126 &65536  ; #3腔体机构自动步序号
LD>=L(326) D1130 &1048576  ; #3腔体机构单检步序号
AND<L(311) D1130 &4194304  ; #3腔体机构单检步序号
ORLD
ANDNOT H5.15  ; 腔体模式（0-正压 1-负压）
ORLD
ANDLD
OUT D1122.13  ; #3腔体机构正常清氦需求（正压测试）
; rung 31
LD P_On
OUT TR0
LD>=L(326) D1176 &8  ; #4腔体机构自动步序号
AND<L(311) D1176 &2048  ; #4腔体机构自动步序号
LD>=L(326) D1180 &8  ; #4腔体机构单检步序号
AND<L(311) D1180 &1024  ; #4腔体机构单检步序号
ORLD
LD>=L(326) D1180 &4096  ; #4腔体机构单检步序号
AND<L(311) D1180 &524288  ; #4腔体机构单检步序号
ORLD
ANDLD
ANDNOT T2605  ; #4-1腔体抽气阀关闭延时（测试）
OUT D1172.12  ; #4腔体机构腔体抽真空需求（测试）
LD TR0
LD>L(321) D1184 &1  ; #4腔体机构清氦步序号
AND H47.00  ; #4腔体有清氦需求
LD>=L(326) D1176 &16384  ; #4腔体机构自动步序号
AND<L(311) D1176 &65536  ; #4腔体机构自动步序号
LD>=L(326) D1180 &1048576  ; #4腔体机构单检步序号
AND<L(311) D1180 &4194304  ; #4腔体机构单检步序号
ORLD
ANDNOT H5.15  ; 腔体模式（0-正压 1-负压）
ORLD
ANDLD
OUT D1172.13  ; #4腔体机构正常清氦需求（正压测试）

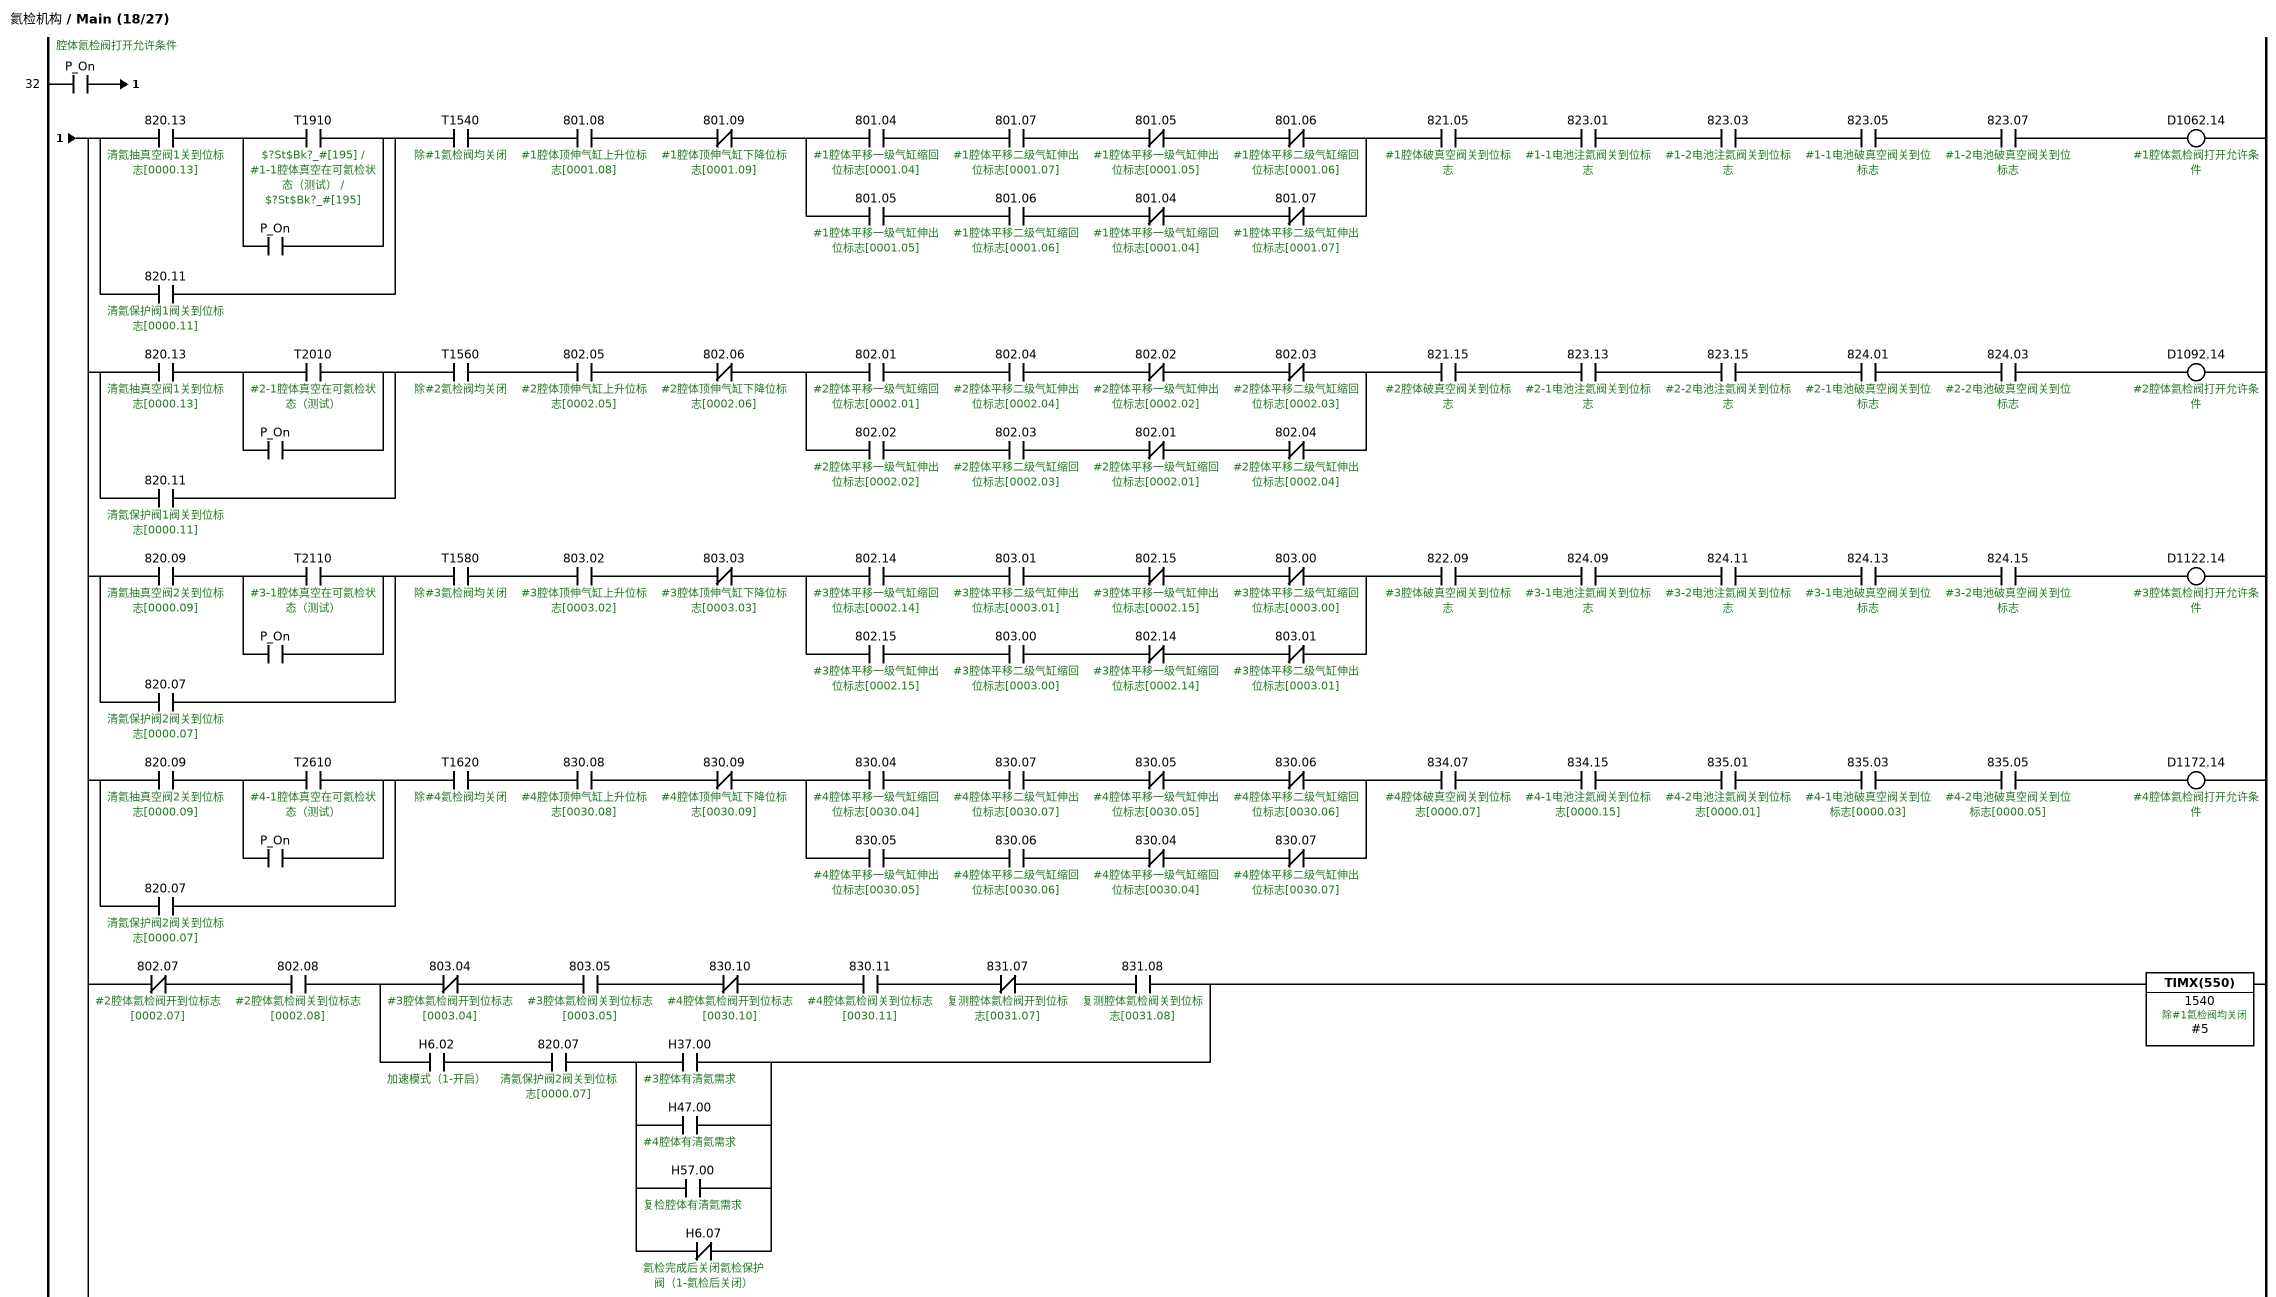

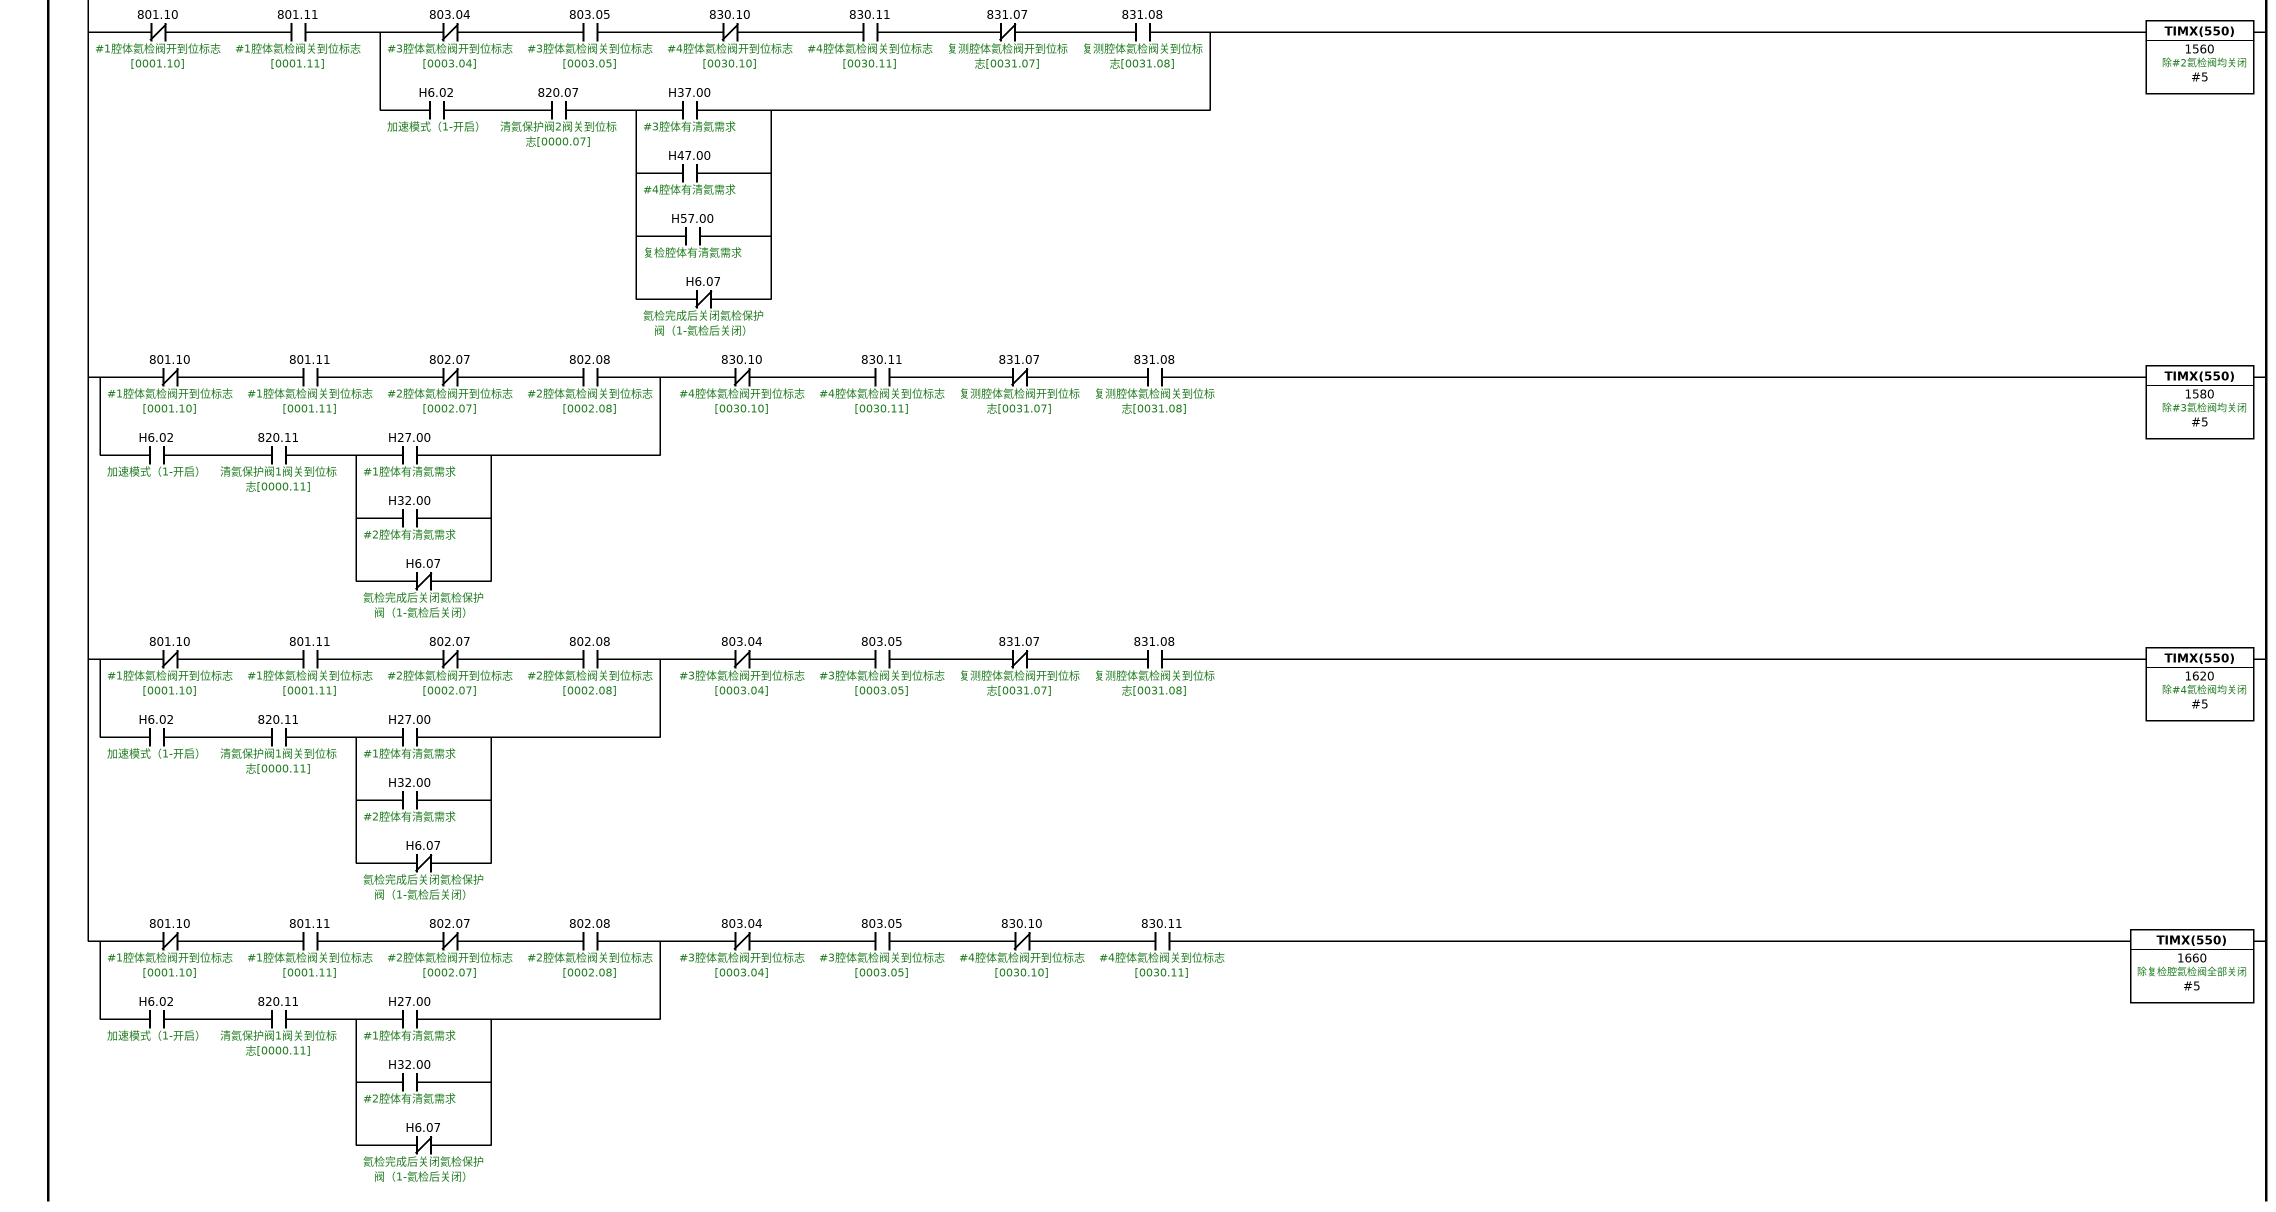
; rung 32: 腔体氦检阀打开允许条件
LD P_On
OUT TR0
LD 820.13  ; 清氦抽真空阀1关到位标志[0000.13]
LD T1910  ; $?St$Bk?_#[195] / #1-1腔体真空在可氦检状态（测试） / $?St$Bk?_#[195]
OR P_On
ANDLD
OR 820.11  ; 清氦保护阀1阀关到位标志[0000.11]
ANDLD
AND T1540  ; 除#1氦检阀均关闭
AND 801.08  ; #1腔体顶伸气缸上升位标志[0001.08]
ANDNOT 801.09  ; #1腔体顶伸气缸下降位标志[0001.09]
LD 801.04  ; #1腔体平移一级气缸缩回位标志[0001.04]
AND 801.07  ; #1腔体平移二级气缸伸出位标志[0001.07]
ANDNOT 801.05  ; #1腔体平移一级气缸伸出位标志[0001.05]
ANDNOT 801.06  ; #1腔体平移二级气缸缩回位标志[0001.06]
LD 801.05  ; #1腔体平移一级气缸伸出位标志[0001.05]
AND 801.06  ; #1腔体平移二级气缸缩回位标志[0001.06]
ANDNOT 801.04  ; #1腔体平移一级气缸缩回位标志[0001.04]
ANDNOT 801.07  ; #1腔体平移二级气缸伸出位标志[0001.07]
ORLD
ANDLD
AND 821.05  ; #1腔体破真空阀关到位标志
AND 823.01  ; #1-1电池注氦阀关到位标志
AND 823.03  ; #1-2电池注氦阀关到位标志
AND 823.05  ; #1-1电池破真空阀关到位标志
AND 823.07  ; #1-2电池破真空阀关到位标志
OUT D1062.14  ; #1腔体氦检阀打开允许条件
LD TR0
LD 820.13  ; 清氦抽真空阀1关到位标志[0000.13]
LD T2010  ; #2-1腔体真空在可氦检状态（测试）
OR P_On
ANDLD
OR 820.11  ; 清氦保护阀1阀关到位标志[0000.11]
ANDLD
AND T1560  ; 除#2氦检阀均关闭
AND 802.05  ; #2腔体顶伸气缸上升位标志[0002.05]
ANDNOT 802.06  ; #2腔体顶伸气缸下降位标志[0002.06]
LD 802.01  ; #2腔体平移一级气缸缩回位标志[0002.01]
AND 802.04  ; #2腔体平移二级气缸伸出位标志[0002.04]
ANDNOT 802.02  ; #2腔体平移一级气缸伸出位标志[0002.02]
ANDNOT 802.03  ; #2腔体平移二级气缸缩回位标志[0002.03]
LD 802.02  ; #2腔体平移一级气缸伸出位标志[0002.02]
AND 802.03  ; #2腔体平移二级气缸缩回位标志[0002.03]
ANDNOT 802.01  ; #2腔体平移一级气缸缩回位标志[0002.01]
ANDNOT 802.04  ; #2腔体平移二级气缸伸出位标志[0002.04]
ORLD
ANDLD
AND 821.15  ; #2腔体破真空阀关到位标志
AND 823.13  ; #2-1电池注氦阀关到位标志
AND 823.15  ; #2-2电池注氦阀关到位标志
AND 824.01  ; #2-1电池破真空阀关到位标志
AND 824.03  ; #2-2电池破真空阀关到位标志
OUT D1092.14  ; #2腔体氦检阀打开允许条件
LD TR0
LD 820.09  ; 清氦抽真空阀2关到位标志[0000.09]
LD T2110  ; #3-1腔体真空在可氦检状态（测试）
OR P_On
ANDLD
OR 820.07  ; 清氦保护阀2阀关到位标志[0000.07]
ANDLD
AND T1580  ; 除#3氦检阀均关闭
AND 803.02  ; #3腔体顶伸气缸上升位标志[0003.02]
ANDNOT 803.03  ; #3腔体顶伸气缸下降位标志[0003.03]
LD 802.14  ; #3腔体平移一级气缸缩回位标志[0002.14]
AND 803.01  ; #3腔体平移二级气缸伸出位标志[0003.01]
ANDNOT 802.15  ; #3腔体平移一级气缸伸出位标志[0002.15]
ANDNOT 803.00  ; #3腔体平移二级气缸缩回位标志[0003.00]
LD 802.15  ; #3腔体平移一级气缸伸出位标志[0002.15]
AND 803.00  ; #3腔体平移二级气缸缩回位标志[0003.00]
ANDNOT 802.14  ; #3腔体平移一级气缸缩回位标志[0002.14]
ANDNOT 803.01  ; #3腔体平移二级气缸伸出位标志[0003.01]
ORLD
ANDLD
AND 822.09  ; #3腔体破真空阀关到位标志
AND 824.09  ; #3-1电池注氦阀关到位标志
AND 824.11  ; #3-2电池注氦阀关到位标志
AND 824.13  ; #3-1电池破真空阀关到位标志
AND 824.15  ; #3-2电池破真空阀关到位标志
OUT D1122.14  ; #3腔体氦检阀打开允许条件
LD TR0
LD 820.09  ; 清氦抽真空阀2关到位标志[0000.09]
LD T2610  ; #4-1腔体真空在可氦检状态（测试）
OR P_On
ANDLD
OR 820.07  ; 清氦保护阀2阀关到位标志[0000.07]
ANDLD
AND T1620  ; 除#4氦检阀均关闭
AND 830.08  ; #4腔体顶伸气缸上升位标志[0030.08]
ANDNOT 830.09  ; #4腔体顶伸气缸下降位标志[0030.09]
LD 830.04  ; #4腔体平移一级气缸缩回位标志[0030.04]
AND 830.07  ; #4腔体平移二级气缸伸出位标志[0030.07]
ANDNOT 830.05  ; #4腔体平移一级气缸伸出位标志[0030.05]
ANDNOT 830.06  ; #4腔体平移二级气缸缩回位标志[0030.06]
LD 830.05  ; #4腔体平移一级气缸伸出位标志[0030.05]
AND 830.06  ; #4腔体平移二级气缸缩回位标志[0030.06]
ANDNOT 830.04  ; #4腔体平移一级气缸缩回位标志[0030.04]
ANDNOT 830.07  ; #4腔体平移二级气缸伸出位标志[0030.07]
ORLD
ANDLD
AND 834.07  ; #4腔体破真空阀关到位标志[0000.07]
AND 834.15  ; #4-1电池注氦阀关到位标志[0000.15]
AND 835.01  ; #4-2电池注氦阀关到位标志[0000.01]
AND 835.03  ; #4-1电池破真空阀关到位标志[0000.03]
AND 835.05  ; #4-2电池破真空阀关到位标志[0000.05]
OUT D1172.14  ; #4腔体氦检阀打开允许条件
LD TR0
ANDNOT 802.07  ; #2腔体氦检阀开到位标志[0002.07]
AND 802.08  ; #2腔体氦检阀关到位标志[0002.08]
LDNOT 803.04  ; #3腔体氦检阀开到位标志[0003.04]
AND 803.05  ; #3腔体氦检阀关到位标志[0003.05]
ANDNOT 830.10  ; #4腔体氦检阀开到位标志[0030.10]
AND 830.11  ; #4腔体氦检阀关到位标志[0030.11]
ANDNOT 831.07  ; 复测腔体氦检阀开到位标志[0031.07]
AND 831.08  ; 复测腔体氦检阀关到位标志[0031.08]
LD H6.02  ; 加速模式（1-开启）
AND 820.07  ; 清氦保护阀2阀关到位标志[0000.07]
LD H37.00  ; #3腔体有清氦需求
OR H47.00  ; #4腔体有清氦需求
OR H57.00  ; 复检腔体有清氦需求
ORNOT H6.07  ; 氦检完成后关闭氦检保护阀（1-氦检后关闭）
ANDLD
ORLD
ANDLD
TIMX(550) 1540 #5  ; 除#1氦检阀均关闭
LD TR0
ANDNOT 801.10  ; #1腔体氦检阀开到位标志[0001.10]
AND 801.11  ; #1腔体氦检阀关到位标志[0001.11]
LDNOT 803.04  ; #3腔体氦检阀开到位标志[0003.04]
AND 803.05  ; #3腔体氦检阀关到位标志[0003.05]
ANDNOT 830.10  ; #4腔体氦检阀开到位标志[0030.10]
AND 830.11  ; #4腔体氦检阀关到位标志[0030.11]
ANDNOT 831.07  ; 复测腔体氦检阀开到位标志[0031.07]
AND 831.08  ; 复测腔体氦检阀关到位标志[0031.08]
LD H6.02  ; 加速模式（1-开启）
AND 820.07  ; 清氦保护阀2阀关到位标志[0000.07]
LD H37.00  ; #3腔体有清氦需求
OR H47.00  ; #4腔体有清氦需求
OR H57.00  ; 复检腔体有清氦需求
ORNOT H6.07  ; 氦检完成后关闭氦检保护阀（1-氦检后关闭）
ANDLD
ORLD
ANDLD
TIMX(550) 1560 #5  ; 除#2氦检阀均关闭
LD TR0
LDNOT 801.10  ; #1腔体氦检阀开到位标志[0001.10]
AND 801.11  ; #1腔体氦检阀关到位标志[0001.11]
ANDNOT 802.07  ; #2腔体氦检阀开到位标志[0002.07]
AND 802.08  ; #2腔体氦检阀关到位标志[0002.08]
LD H6.02  ; 加速模式（1-开启）
AND 820.11  ; 清氦保护阀1阀关到位标志[0000.11]
LD H27.00  ; #1腔体有清氦需求
OR H32.00  ; #2腔体有清氦需求
ORNOT H6.07  ; 氦检完成后关闭氦检保护阀（1-氦检后关闭）
ANDLD
ORLD
ANDLD
ANDNOT 830.10  ; #4腔体氦检阀开到位标志[0030.10]
AND 830.11  ; #4腔体氦检阀关到位标志[0030.11]
ANDNOT 831.07  ; 复测腔体氦检阀开到位标志[0031.07]
AND 831.08  ; 复测腔体氦检阀关到位标志[0031.08]
TIMX(550) 1580 #5  ; 除#3氦检阀均关闭
LD TR0
LDNOT 801.10  ; #1腔体氦检阀开到位标志[0001.10]
AND 801.11  ; #1腔体氦检阀关到位标志[0001.11]
ANDNOT 802.07  ; #2腔体氦检阀开到位标志[0002.07]
AND 802.08  ; #2腔体氦检阀关到位标志[0002.08]
LD H6.02  ; 加速模式（1-开启）
AND 820.11  ; 清氦保护阀1阀关到位标志[0000.11]
LD H27.00  ; #1腔体有清氦需求
OR H32.00  ; #2腔体有清氦需求
ORNOT H6.07  ; 氦检完成后关闭氦检保护阀（1-氦检后关闭）
ANDLD
ORLD
ANDLD
ANDNOT 803.04  ; #3腔体氦检阀开到位标志[0003.04]
AND 803.05  ; #3腔体氦检阀关到位标志[0003.05]
ANDNOT 831.07  ; 复测腔体氦检阀开到位标志[0031.07]
AND 831.08  ; 复测腔体氦检阀关到位标志[0031.08]
TIMX(550) 1620 #5  ; 除#4氦检阀均关闭
LD TR0
LDNOT 801.10  ; #1腔体氦检阀开到位标志[0001.10]
AND 801.11  ; #1腔体氦检阀关到位标志[0001.11]
ANDNOT 802.07  ; #2腔体氦检阀开到位标志[0002.07]
AND 802.08  ; #2腔体氦检阀关到位标志[0002.08]
LD H6.02  ; 加速模式（1-开启）
AND 820.11  ; 清氦保护阀1阀关到位标志[0000.11]
LD H27.00  ; #1腔体有清氦需求
OR H32.00  ; #2腔体有清氦需求
ORNOT H6.07  ; 氦检完成后关闭氦检保护阀（1-氦检后关闭）
ANDLD
ORLD
ANDLD
ANDNOT 803.04  ; #3腔体氦检阀开到位标志[0003.04]
AND 803.05  ; #3腔体氦检阀关到位标志[0003.05]
ANDNOT 830.10  ; #4腔体氦检阀开到位标志[0030.10]
AND 830.11  ; #4腔体氦检阀关到位标志[0030.11]
TIMX(550) 1660 #5  ; 除复检腔氦检阀全部关闭

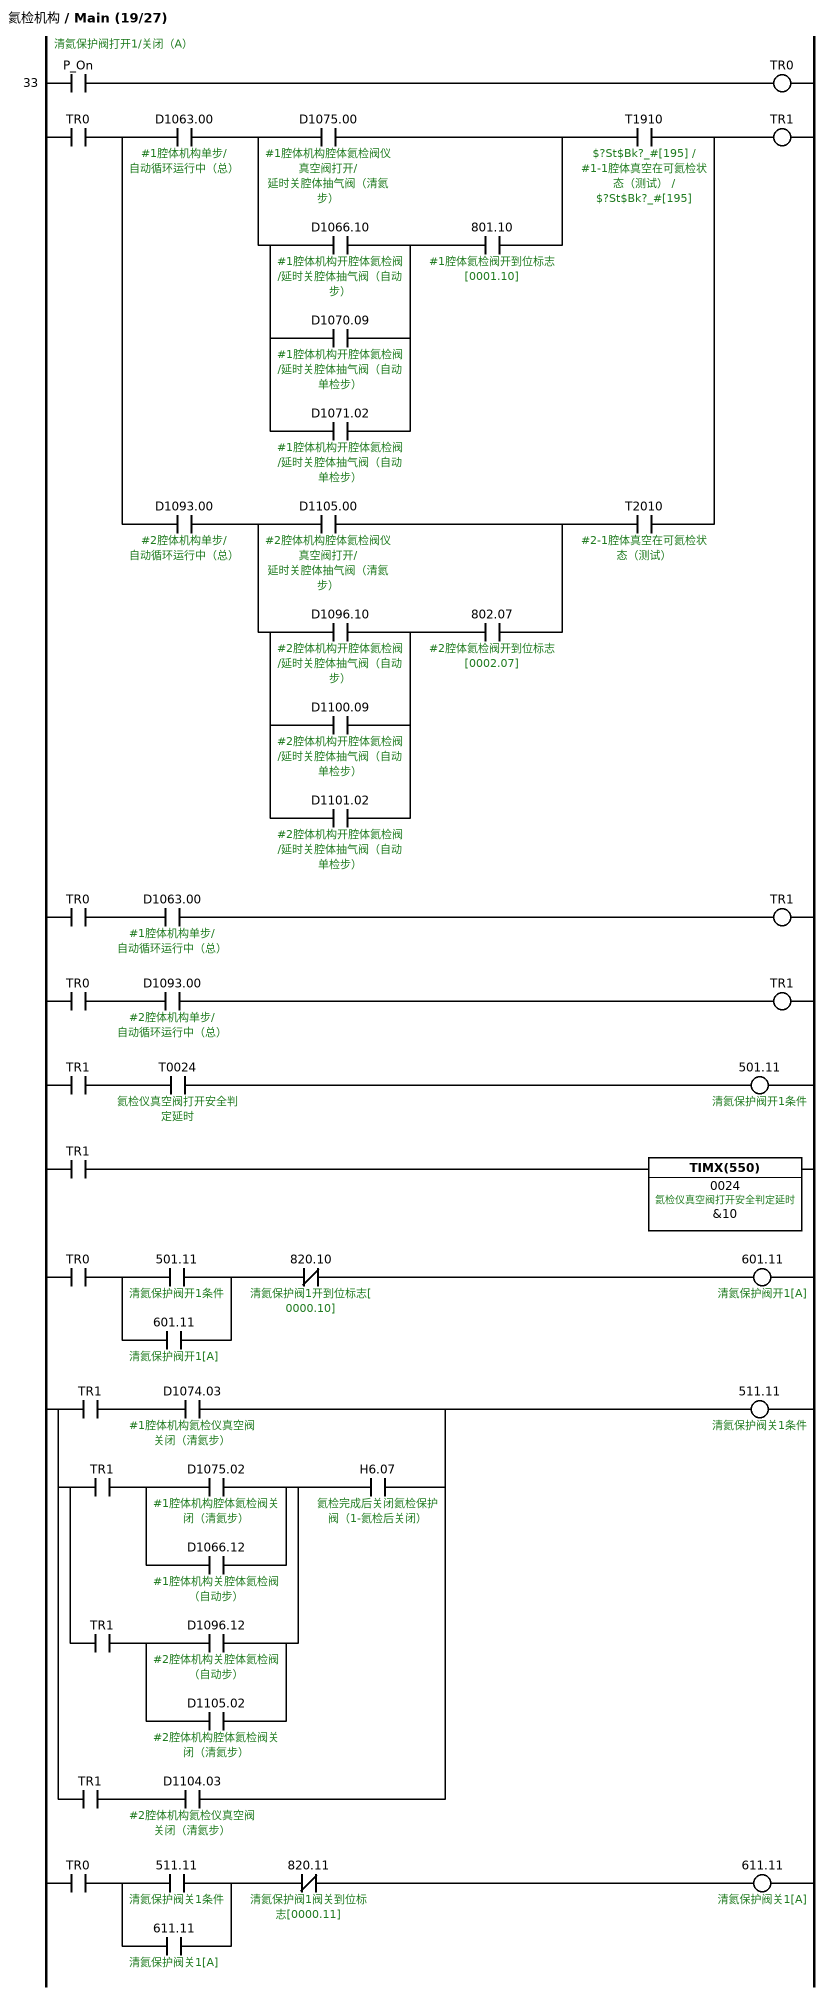
; rung 33: 清氦保护阀打开1/关闭（A）
LD P_On
OUT TR0
LD D1063.00  ; #1腔体机构单步/自动循环运行中（总）
LD D1075.00  ; #1腔体机构腔体氦检阀仪真空阀打开/延时关腔体抽气阀（清氦步）
LD D1066.10  ; #1腔体机构开腔体氦检阀/延时关腔体抽气阀（自动步）
OR D1070.09  ; #1腔体机构开腔体氦检阀/延时关腔体抽气阀（自动单检步）
OR D1071.02  ; #1腔体机构开腔体氦检阀/延时关腔体抽气阀（自动单检步）
AND 801.10  ; #1腔体氦检阀开到位标志[0001.10]
ORLD
ANDLD
AND T1910  ; $?St$Bk?_#[195] / #1-1腔体真空在可氦检状态（测试） / $?St$Bk?_#[195]
LD D1093.00  ; #2腔体机构单步/自动循环运行中（总）
LD D1105.00  ; #2腔体机构腔体氦检阀仪真空阀打开/延时关腔体抽气阀（清氦步）
LD D1096.10  ; #2腔体机构开腔体氦检阀/延时关腔体抽气阀（自动步）
OR D1100.09  ; #2腔体机构开腔体氦检阀/延时关腔体抽气阀（自动单检步）
OR D1101.02  ; #2腔体机构开腔体氦检阀/延时关腔体抽气阀（自动单检步）
AND 802.07  ; #2腔体氦检阀开到位标志[0002.07]
ORLD
ANDLD
AND T2010  ; #2-1腔体真空在可氦检状态（测试）
ORLD
ANDLD
OUT TR1
AND T0024  ; 氦检仪真空阀打开安全判定延时
OUT 501.11  ; 清氦保护阀开1条件
LD TR1
TIMX(550) 0024 &10  ; 氦检仪真空阀打开安全判定延时
LD TR0
LD 501.11  ; 清氦保护阀开1条件
OR 601.11  ; 清氦保护阀开1[A]
ANDLD
ANDNOT 820.10  ; 清氦保护阀1开到位标志[0000.10]
OUT 601.11  ; 清氦保护阀开1[A]
LD TR0
AND D1063.00  ; #1腔体机构单步/自动循环运行中（总）
OUT TR1
AND D1074.03  ; #1腔体机构氦检仪真空阀关闭（清氦步）
LD TR1
LD D1075.02  ; #1腔体机构腔体氦检阀关闭（清氦步）
OR D1066.12  ; #1腔体机构关腔体氦检阀（自动步）
ANDLD
LD TR0
AND D1093.00  ; #2腔体机构单步/自动循环运行中（总）
OUT TR1
LD D1096.12  ; #2腔体机构关腔体氦检阀（自动步）
OR D1105.02  ; #2腔体机构腔体氦检阀关闭（清氦步）
ANDLD
ORLD
AND H6.07  ; 氦检完成后关闭氦检保护阀（1-氦检后关闭）
ORLD
LD TR1
AND D1104.03  ; #2腔体机构氦检仪真空阀关闭（清氦步）
ORLD
OUT 511.11  ; 清氦保护阀关1条件
LD TR0
LD 511.11  ; 清氦保护阀关1条件
OR 611.11  ; 清氦保护阀关1[A]
ANDLD
ANDNOT 820.11  ; 清氦保护阀1阀关到位标志[0000.11]
OUT 611.11  ; 清氦保护阀关1[A]

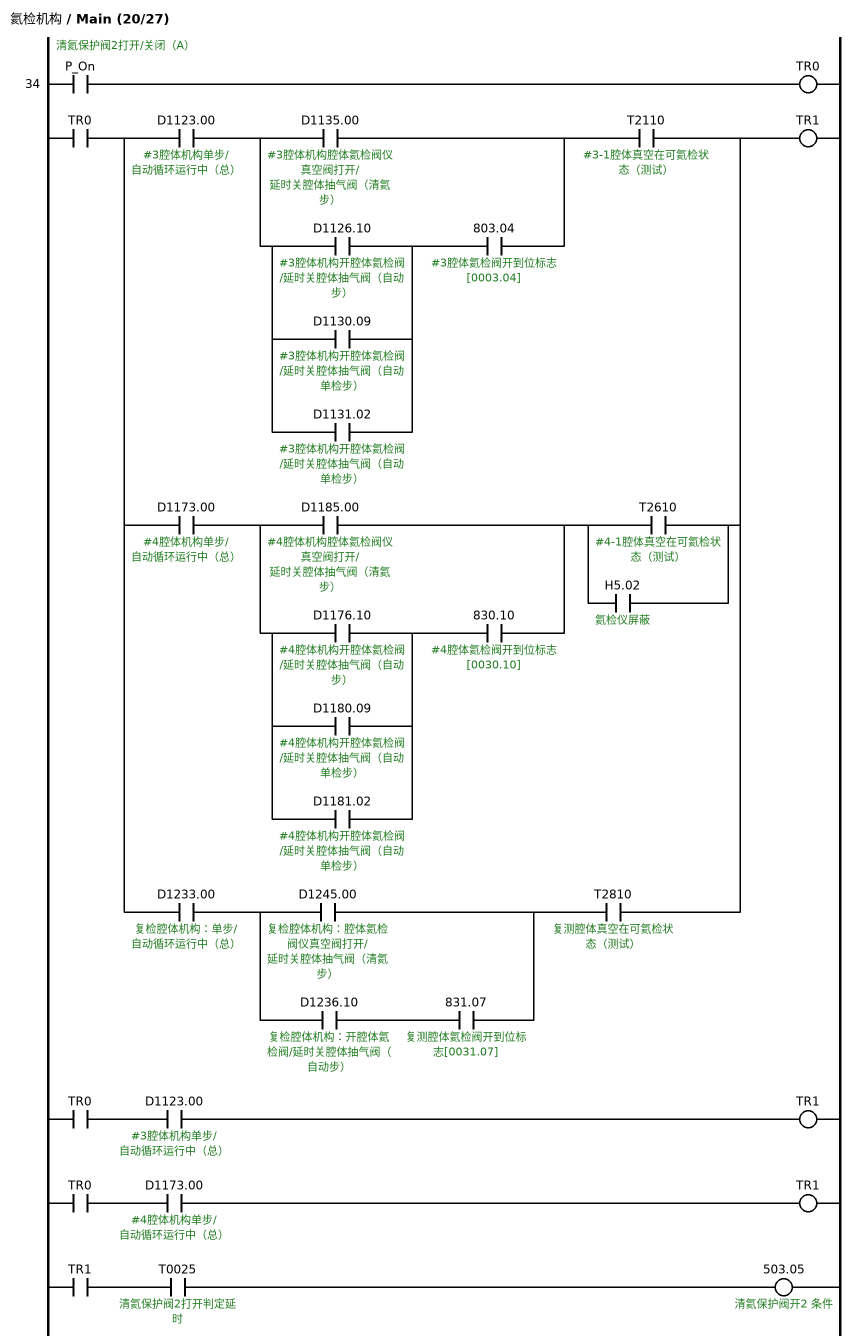

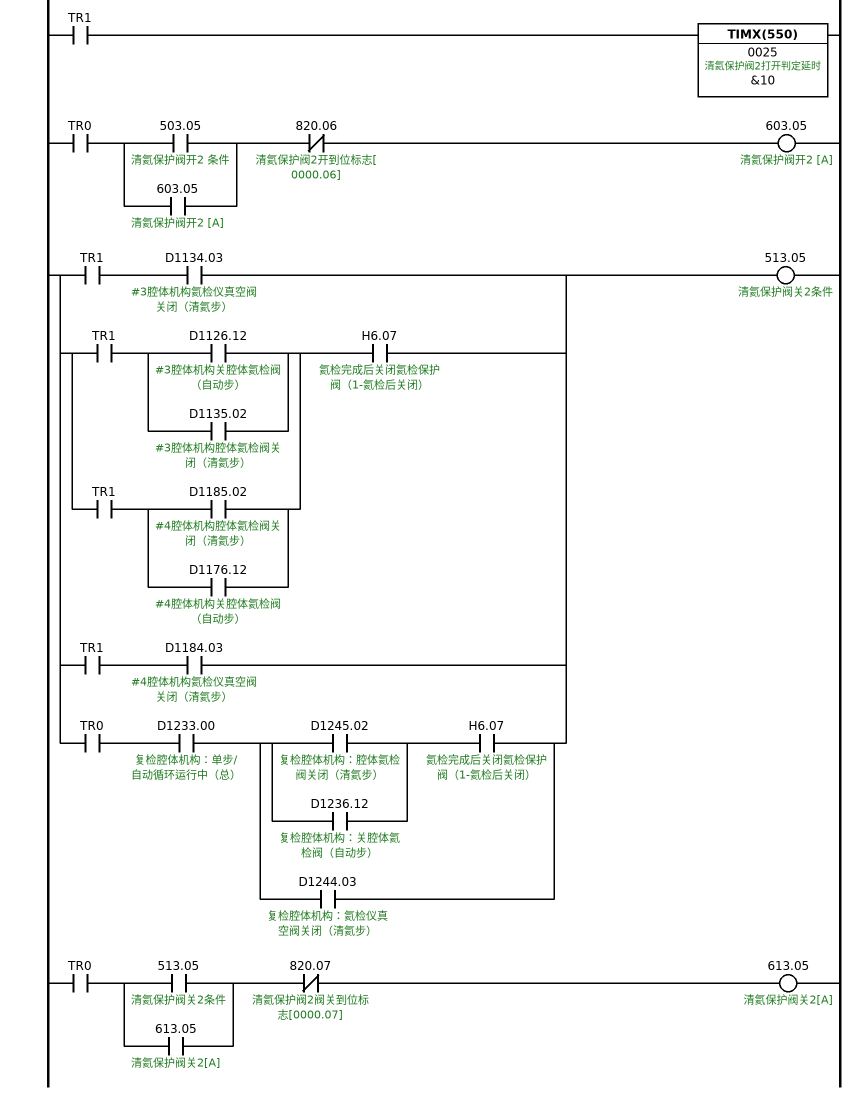
; rung 34: 清氦保护阀2打开/关闭（A）
LD P_On
OUT TR0
LD D1123.00  ; #3腔体机构单步/自动循环运行中（总）
LD D1135.00  ; #3腔体机构腔体氦检阀仪真空阀打开/延时关腔体抽气阀（清氦步）
LD D1126.10  ; #3腔体机构开腔体氦检阀/延时关腔体抽气阀（自动步）
OR D1130.09  ; #3腔体机构开腔体氦检阀/延时关腔体抽气阀（自动单检步）
OR D1131.02  ; #3腔体机构开腔体氦检阀/延时关腔体抽气阀（自动单检步）
AND 803.04  ; #3腔体氦检阀开到位标志[0003.04]
ORLD
ANDLD
AND T2110  ; #3-1腔体真空在可氦检状态（测试）
LD D1173.00  ; #4腔体机构单步/自动循环运行中（总）
LD D1185.00  ; #4腔体机构腔体氦检阀仪真空阀打开/延时关腔体抽气阀（清氦步）
LD D1176.10  ; #4腔体机构开腔体氦检阀/延时关腔体抽气阀（自动步）
OR D1180.09  ; #4腔体机构开腔体氦检阀/延时关腔体抽气阀（自动单检步）
OR D1181.02  ; #4腔体机构开腔体氦检阀/延时关腔体抽气阀（自动单检步）
AND 830.10  ; #4腔体氦检阀开到位标志[0030.10]
ORLD
ANDLD
LD T2610  ; #4-1腔体真空在可氦检状态（测试）
OR H5.02  ; 氦检仪屏蔽
ANDLD
ORLD
LD D1233.00  ; 复检腔体机构：单步/自动循环运行中（总）
LD D1245.00  ; 复检腔体机构：腔体氦检阀仪真空阀打开/延时关腔体抽气阀（清氦步）
LD D1236.10  ; 复检腔体机构：开腔体氦检阀/延时关腔体抽气阀（自动步）
AND 831.07  ; 复测腔体氦检阀开到位标志[0031.07]
ORLD
ANDLD
AND T2810  ; 复测腔体真空在可氦检状态（测试）
ORLD
ANDLD
OUT TR1
AND T0025  ; 清氦保护阀2打开判定延时
OUT 503.05  ; 清氦保护阀开2 条件
LD TR1
TIMX(550) 0025 &10  ; 清氦保护阀2打开判定延时
LD TR0
LD 503.05  ; 清氦保护阀开2 条件
OR 603.05  ; 清氦保护阀开2 [A]
ANDLD
ANDNOT 820.06  ; 清氦保护阀2开到位标志[0000.06]
OUT 603.05  ; 清氦保护阀开2 [A]
LD TR0
AND D1123.00  ; #3腔体机构单步/自动循环运行中（总）
OUT TR1
AND D1134.03  ; #3腔体机构氦检仪真空阀关闭（清氦步）
LD TR1
LD D1126.12  ; #3腔体机构关腔体氦检阀（自动步）
OR D1135.02  ; #3腔体机构腔体氦检阀关闭（清氦步）
ANDLD
LD TR0
AND D1173.00  ; #4腔体机构单步/自动循环运行中（总）
OUT TR1
LD D1185.02  ; #4腔体机构腔体氦检阀关闭（清氦步）
OR D1176.12  ; #4腔体机构关腔体氦检阀（自动步）
ANDLD
ORLD
AND H6.07  ; 氦检完成后关闭氦检保护阀（1-氦检后关闭）
ORLD
LD TR1
AND D1184.03  ; #4腔体机构氦检仪真空阀关闭（清氦步）
LD TR0
AND D1233.00  ; 复检腔体机构：单步/自动循环运行中（总）
LD D1245.02  ; 复检腔体机构：腔体氦检阀关闭（清氦步）
OR D1236.12  ; 复检腔体机构：关腔体氦检阀（自动步）
AND H6.07  ; 氦检完成后关闭氦检保护阀（1-氦检后关闭）
OR D1244.03  ; 复检腔体机构：氦检仪真空阀关闭（清氦步）
ANDLD
ORLD
ORLD
OUT 513.05  ; 清氦保护阀关2条件
LD TR0
LD 513.05  ; 清氦保护阀关2条件
OR 613.05  ; 清氦保护阀关2[A]
ANDLD
ANDNOT 820.07  ; 清氦保护阀2阀关到位标志[0000.07]
OUT 613.05  ; 清氦保护阀关2[A]

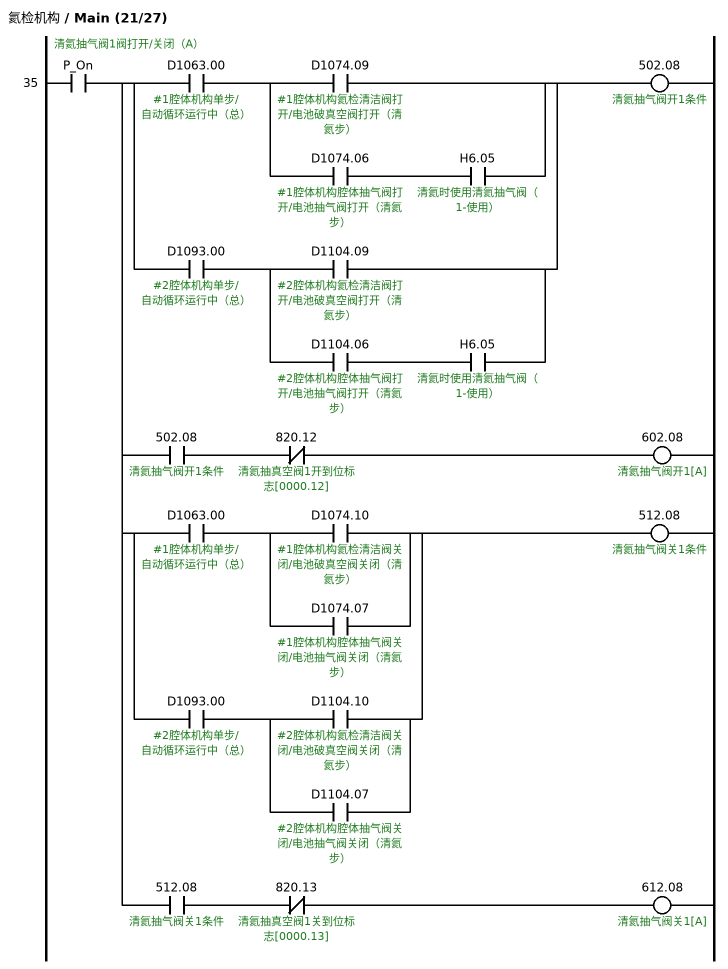
; rung 35: 清氦抽气阀1阀打开/关闭（A）
LD P_On
OUT TR0
LD D1063.00  ; #1腔体机构单步/自动循环运行中（总）
LD D1074.09  ; #1腔体机构氦检清洁阀打开/电池破真空阀打开（清氦步）
LD D1074.06  ; #1腔体机构腔体抽气阀打开/电池抽气阀打开（清氦步）
AND H6.05  ; 清氦时使用清氦抽气阀（1-使用）
ORLD
ANDLD
LD D1093.00  ; #2腔体机构单步/自动循环运行中（总）
LD D1104.09  ; #2腔体机构氦检清洁阀打开/电池破真空阀打开（清氦步）
LD D1104.06  ; #2腔体机构腔体抽气阀打开/电池抽气阀打开（清氦步）
AND H6.05  ; 清氦时使用清氦抽气阀（1-使用）
ORLD
ANDLD
ORLD
ANDLD
OUT 502.08  ; 清氦抽气阀开1条件
LD TR0
AND 502.08  ; 清氦抽气阀开1条件
ANDNOT 820.12  ; 清氦抽真空阀1开到位标志[0000.12]
OUT 602.08  ; 清氦抽气阀开1[A]
LD TR0
LD D1063.00  ; #1腔体机构单步/自动循环运行中（总）
LD D1074.10  ; #1腔体机构氦检清洁阀关闭/电池破真空阀关闭（清氦步）
OR D1074.07  ; #1腔体机构腔体抽气阀关闭/电池抽气阀关闭（清氦步）
ANDLD
LD D1093.00  ; #2腔体机构单步/自动循环运行中（总）
LD D1104.10  ; #2腔体机构氦检清洁阀关闭/电池破真空阀关闭（清氦步）
OR D1104.07  ; #2腔体机构腔体抽气阀关闭/电池抽气阀关闭（清氦步）
ANDLD
ORLD
ANDLD
OUT 512.08  ; 清氦抽气阀关1条件
LD TR0
AND 512.08  ; 清氦抽气阀关1条件
ANDNOT 820.13  ; 清氦抽真空阀1关到位标志[0000.13]
OUT 612.08  ; 清氦抽气阀关1[A]

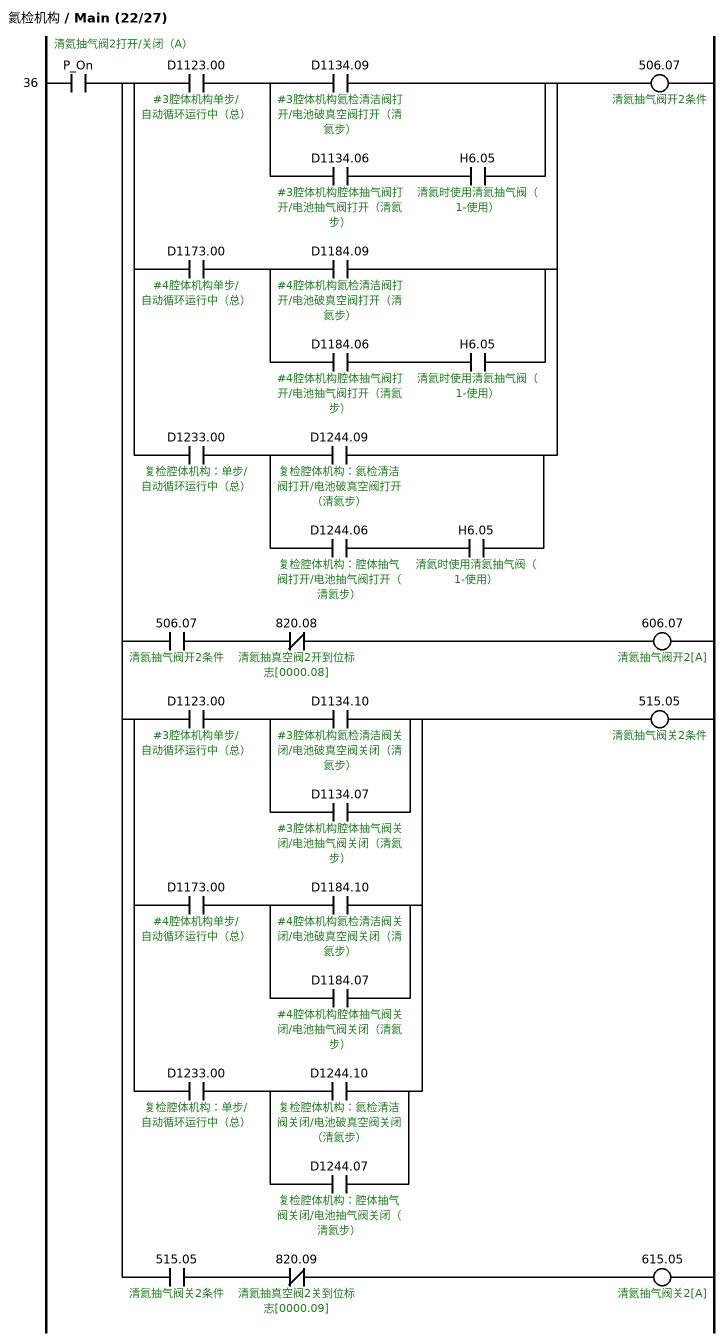
; rung 36: 清氦抽气阀2打开/关闭（A）
LD P_On
OUT TR0
LD D1123.00  ; #3腔体机构单步/自动循环运行中（总）
LD D1134.09  ; #3腔体机构氦检清洁阀打开/电池破真空阀打开（清氦步）
LD D1134.06  ; #3腔体机构腔体抽气阀打开/电池抽气阀打开（清氦步）
AND H6.05  ; 清氦时使用清氦抽气阀（1-使用）
ORLD
ANDLD
LD D1173.00  ; #4腔体机构单步/自动循环运行中（总）
LD D1184.09  ; #4腔体机构氦检清洁阀打开/电池破真空阀打开（清氦步）
LD D1184.06  ; #4腔体机构腔体抽气阀打开/电池抽气阀打开（清氦步）
AND H6.05  ; 清氦时使用清氦抽气阀（1-使用）
ORLD
ANDLD
ORLD
LD D1233.00  ; 复检腔体机构：单步/自动循环运行中（总）
LD D1244.09  ; 复检腔体机构：氦检清洁阀打开/电池破真空阀打开（清氦步）
LD D1244.06  ; 复检腔体机构：腔体抽气阀打开/电池抽气阀打开（清氦步）
AND H6.05  ; 清氦时使用清氦抽气阀（1-使用）
ORLD
ANDLD
ORLD
ANDLD
OUT 506.07  ; 清氦抽气阀开2条件
LD TR0
AND 506.07  ; 清氦抽气阀开2条件
ANDNOT 820.08  ; 清氦抽真空阀2开到位标志[0000.08]
OUT 606.07  ; 清氦抽气阀开2[A]
LD TR0
LD D1123.00  ; #3腔体机构单步/自动循环运行中（总）
LD D1134.10  ; #3腔体机构氦检清洁阀关闭/电池破真空阀关闭（清氦步）
OR D1134.07  ; #3腔体机构腔体抽气阀关闭/电池抽气阀关闭（清氦步）
ANDLD
LD D1173.00  ; #4腔体机构单步/自动循环运行中（总）
LD D1184.10  ; #4腔体机构氦检清洁阀关闭/电池破真空阀关闭（清氦步）
OR D1184.07  ; #4腔体机构腔体抽气阀关闭/电池抽气阀关闭（清氦步）
ANDLD
ORLD
LD D1233.00  ; 复检腔体机构：单步/自动循环运行中（总）
LD D1244.10  ; 复检腔体机构：氦检清洁阀关闭/电池破真空阀关闭（清氦步）
OR D1244.07  ; 复检腔体机构：腔体抽气阀关闭/电池抽气阀关闭（清氦步）
ANDLD
ORLD
ANDLD
OUT 515.05  ; 清氦抽气阀关2条件
LD TR0
AND 515.05  ; 清氦抽气阀关2条件
ANDNOT 820.09  ; 清氦抽真空阀2关到位标志[0000.09]
OUT 615.05  ; 清氦抽气阀关2[A]

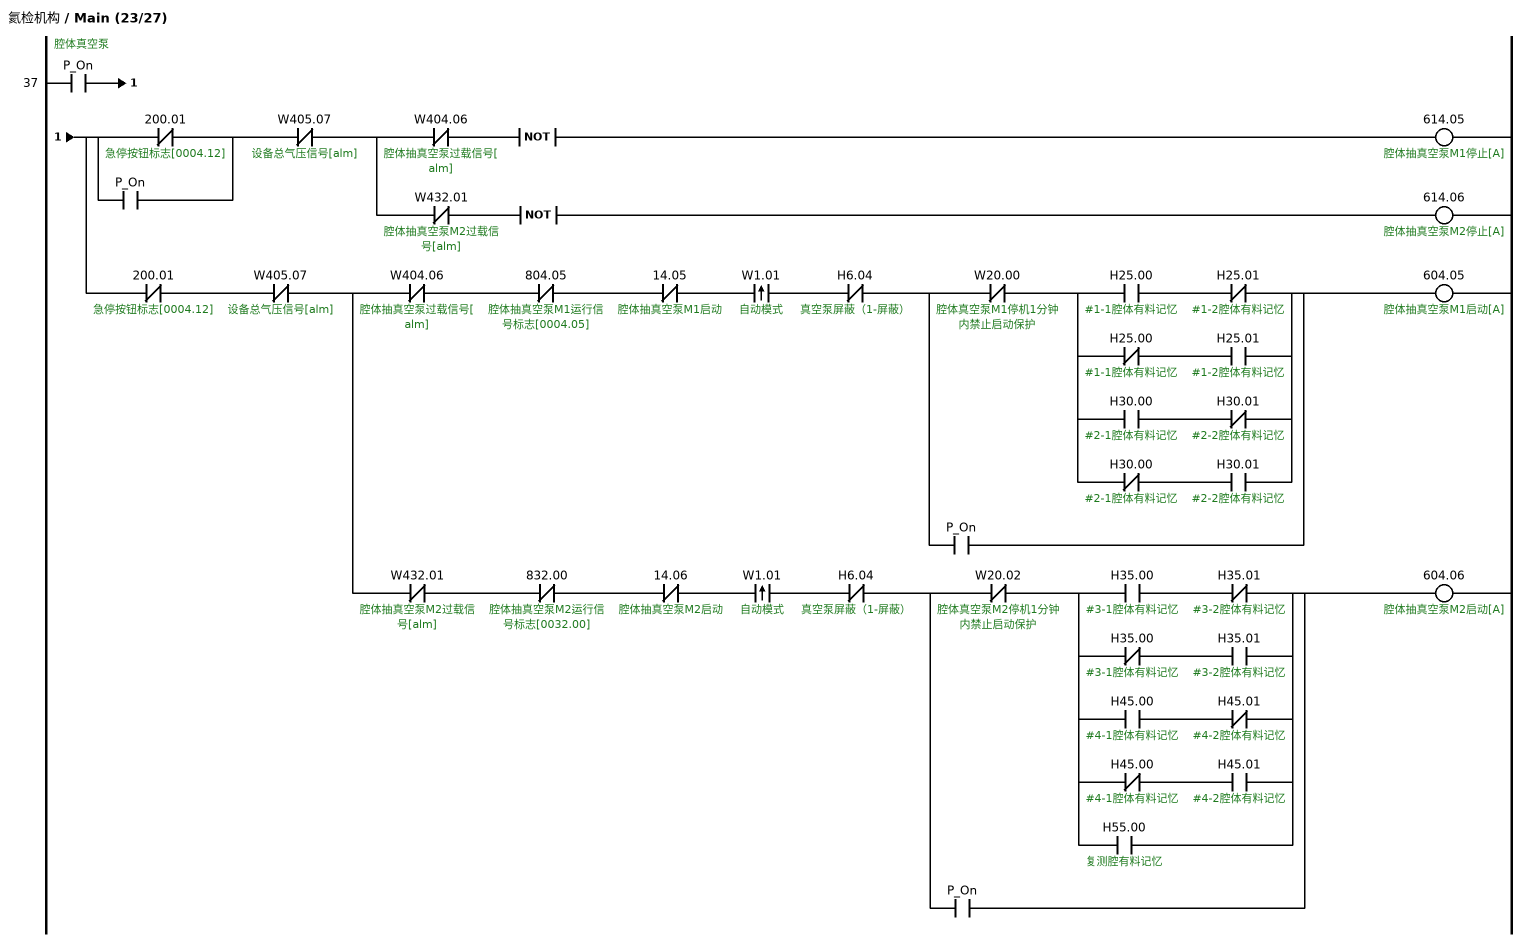
; rung 37: 腔体真空泵
LD P_On
OUT TR0
LDNOT 200.01  ; 急停按钮标志[0004.12]
OR P_On
ANDLD
ANDNOT W405.07  ; 设备总气压信号[alm]
OUT TR1
ANDNOT W404.06  ; 腔体抽真空泵过载信号[alm]
NOT(520)
OUT 614.05  ; 腔体抽真空泵M1停止[A]
LD TR1
ANDNOT W432.01  ; 腔体抽真空泵M2过载信号[alm]
NOT(520)
OUT 614.06  ; 腔体抽真空泵M2停止[A]
LD TR0
ANDNOT 200.01  ; 急停按钮标志[0004.12]
ANDNOT W405.07  ; 设备总气压信号[alm]
OUT TR0
ANDNOT W404.06  ; 腔体抽真空泵过载信号[alm]
ANDNOT 804.05  ; 腔体抽真空泵M1运行信号标志[0004.05]
ANDNOT 14.05  ; 腔体抽真空泵M1启动
@AND W1.01  ; 自动模式
ANDNOT H6.04  ; 真空泵屏蔽（1-屏蔽）
LDNOT W20.00  ; 腔体真空泵M1停机1分钟内禁止启动保护
LD H25.00  ; #1-1腔体有料记忆
ANDNOT H25.01  ; #1-2腔体有料记忆
LDNOT H25.00  ; #1-1腔体有料记忆
AND H25.01  ; #1-2腔体有料记忆
ORLD
LD H30.00  ; #2-1腔体有料记忆
ANDNOT H30.01  ; #2-2腔体有料记忆
ORLD
LDNOT H30.00  ; #2-1腔体有料记忆
AND H30.01  ; #2-2腔体有料记忆
ORLD
ANDLD
OR P_On
ANDLD
OUT 604.05  ; 腔体抽真空泵M1启动[A]
LD TR0
ANDNOT W432.01  ; 腔体抽真空泵M2过载信号[alm]
ANDNOT 832.00  ; 腔体抽真空泵M2运行信号标志[0032.00]
ANDNOT 14.06  ; 腔体抽真空泵M2启动
@AND W1.01  ; 自动模式
ANDNOT H6.04  ; 真空泵屏蔽（1-屏蔽）
LDNOT W20.02  ; 腔体真空泵M2停机1分钟内禁止启动保护
LD H35.00  ; #3-1腔体有料记忆
ANDNOT H35.01  ; #3-2腔体有料记忆
LDNOT H35.00  ; #3-1腔体有料记忆
AND H35.01  ; #3-2腔体有料记忆
ORLD
LD H45.00  ; #4-1腔体有料记忆
ANDNOT H45.01  ; #4-2腔体有料记忆
ORLD
LDNOT H45.00  ; #4-1腔体有料记忆
AND H45.01  ; #4-2腔体有料记忆
ORLD
OR H55.00  ; 复测腔有料记忆
ANDLD
OR P_On
ANDLD
OUT 604.06  ; 腔体抽真空泵M2启动[A]

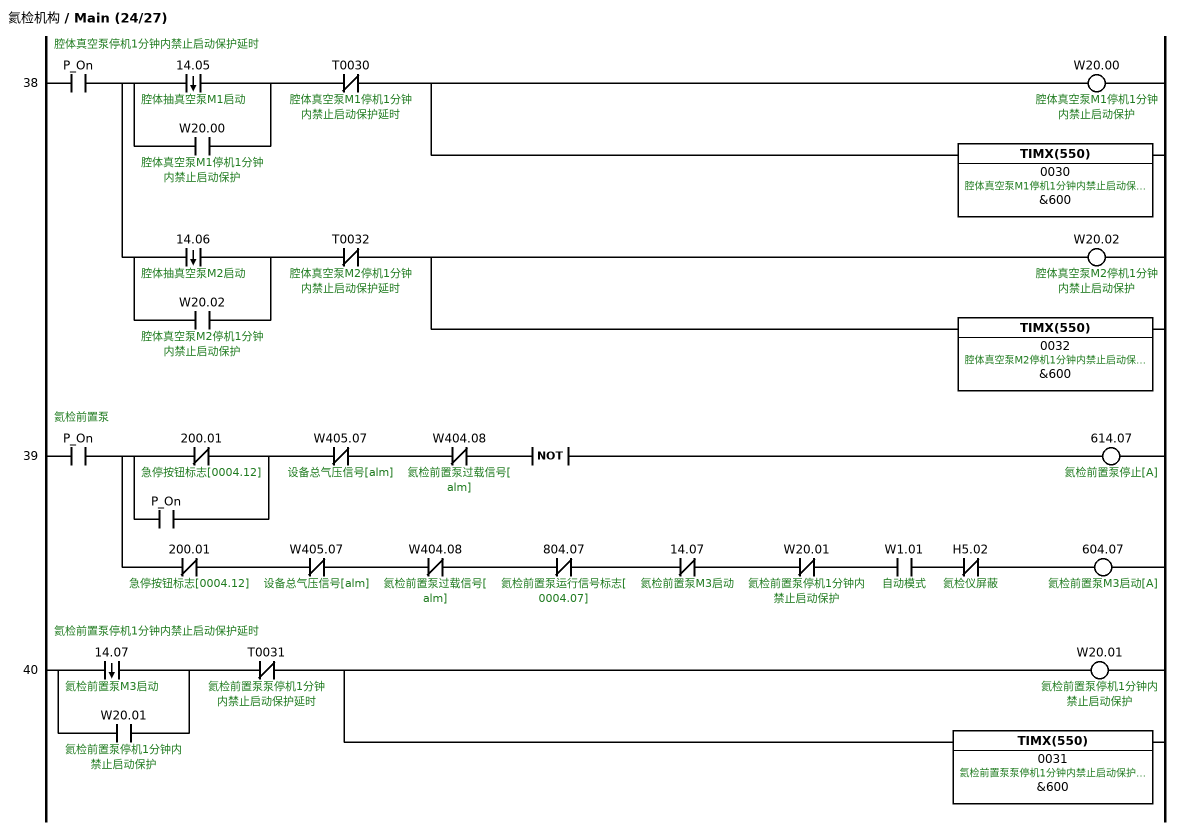
; rung 38: 腔体真空泵停机1分钟内禁止启动保护延时
LD P_On
OUT TR0
%LD 14.05  ; 腔体抽真空泵M1启动
OR W20.00  ; 腔体真空泵M1停机1分钟内禁止启动保护
ANDLD
ANDNOT T0030  ; 腔体真空泵M1停机1分钟内禁止启动保护延时
OUT W20.00  ; 腔体真空泵M1停机1分钟内禁止启动保护
TIMX(550) 0030 &600  ; 腔体真空泵M1停机1分钟内禁止启动保护延时
LD TR0
%LD 14.06  ; 腔体抽真空泵M2启动
OR W20.02  ; 腔体真空泵M2停机1分钟内禁止启动保护
ANDLD
ANDNOT T0032  ; 腔体真空泵M2停机1分钟内禁止启动保护延时
OUT W20.02  ; 腔体真空泵M2停机1分钟内禁止启动保护
TIMX(550) 0032 &600  ; 腔体真空泵M2停机1分钟内禁止启动保护延时
; rung 39: 氦检前置泵
LD P_On
OUT TR0
LDNOT 200.01  ; 急停按钮标志[0004.12]
OR P_On
ANDLD
ANDNOT W405.07  ; 设备总气压信号[alm]
ANDNOT W404.08  ; 氦检前置泵过载信号[alm]
NOT(520)
OUT 614.07  ; 氦检前置泵停止[A]
LD TR0
ANDNOT 200.01  ; 急停按钮标志[0004.12]
ANDNOT W405.07  ; 设备总气压信号[alm]
ANDNOT W404.08  ; 氦检前置泵过载信号[alm]
ANDNOT 804.07  ; 氦检前置泵运行信号标志[0004.07]
ANDNOT 14.07  ; 氦检前置泵M3启动
ANDNOT W20.01  ; 氦检前置泵停机1分钟内禁止启动保护
AND W1.01  ; 自动模式
ANDNOT H5.02  ; 氦检仪屏蔽
OUT 604.07  ; 氦检前置泵M3启动[A]
; rung 40: 氦检前置泵停机1分钟内禁止启动保护延时
%LD 14.07  ; 氦检前置泵M3启动
OR W20.01  ; 氦检前置泵停机1分钟内禁止启动保护
ANDNOT T0031  ; 氦检前置泵泵停机1分钟内禁止启动保护延时
OUT W20.01  ; 氦检前置泵停机1分钟内禁止启动保护
TIMX(550) 0031 &600  ; 氦检前置泵泵停机1分钟内禁止启动保护延时

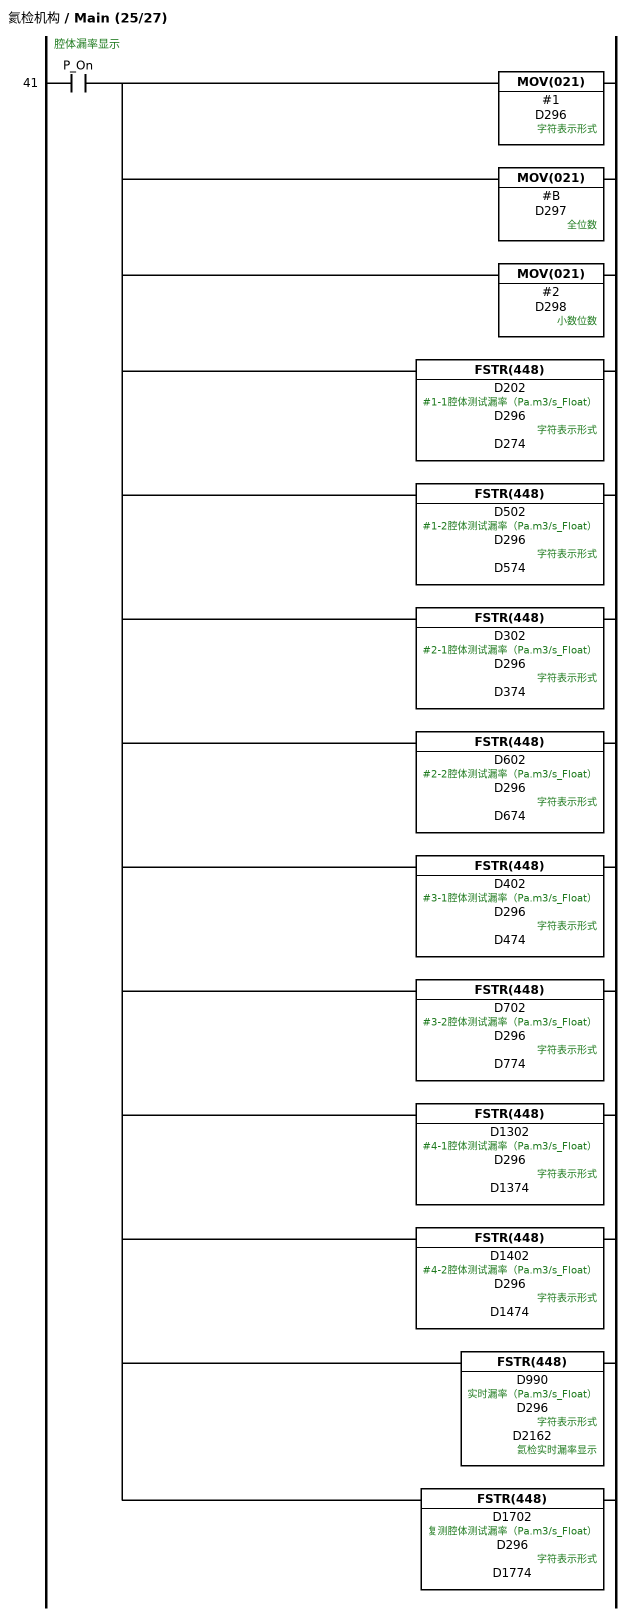
; rung 41: 腔体漏率显示
LD P_On
MOV(021) #1 D296  ; 字符表示形式
MOV(021) #B D297  ; 全位数
MOV(021) #2 D298  ; 小数位数
FSTR(448) D202 D296 D274  ; #1-1腔体测试漏率（Pa.m3/s_Float）, 字符表示形式
FSTR(448) D502 D296 D574  ; #1-2腔体测试漏率（Pa.m3/s_Float）, 字符表示形式
FSTR(448) D302 D296 D374  ; #2-1腔体测试漏率（Pa.m3/s_Float）, 字符表示形式
FSTR(448) D602 D296 D674  ; #2-2腔体测试漏率（Pa.m3/s_Float）, 字符表示形式
FSTR(448) D402 D296 D474  ; #3-1腔体测试漏率（Pa.m3/s_Float）, 字符表示形式
FSTR(448) D702 D296 D774  ; #3-2腔体测试漏率（Pa.m3/s_Float）, 字符表示形式
FSTR(448) D1302 D296 D1374  ; #4-1腔体测试漏率（Pa.m3/s_Float）, 字符表示形式
FSTR(448) D1402 D296 D1474  ; #4-2腔体测试漏率（Pa.m3/s_Float）, 字符表示形式
FSTR(448) D990 D296 D2162  ; 实时漏率（Pa.m3/s_Float）, 字符表示形式, 氦检实时漏率显示
FSTR(448) D1702 D296 D1774  ; 复测腔体测试漏率（Pa.m3/s_Float）, 字符表示形式

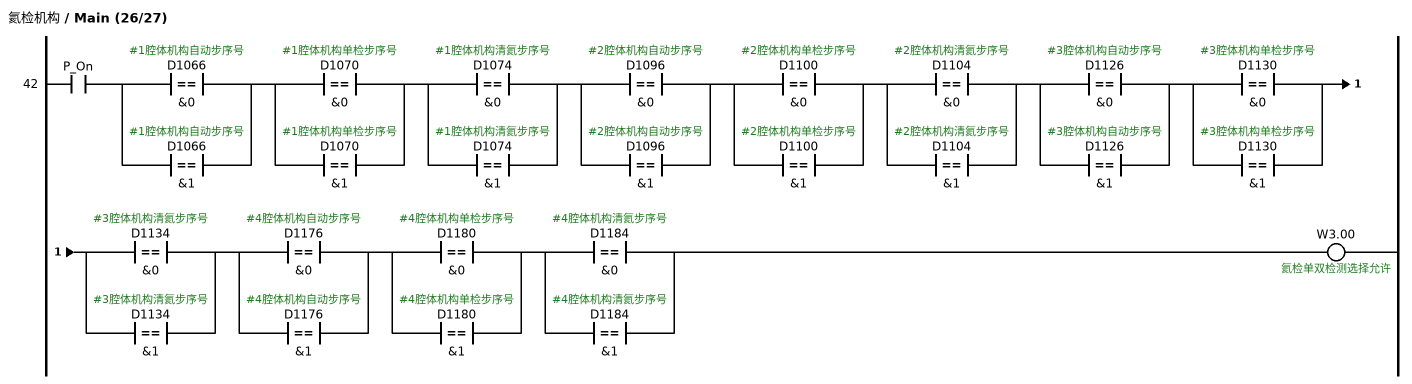
; rung 42
LD P_On
LD=L(301) D1066 &0  ; #1腔体机构自动步序号
OR=L(301) D1066 &1  ; #1腔体机构自动步序号
ANDLD
LD=L(301) D1070 &0  ; #1腔体机构单检步序号
OR=L(301) D1070 &1  ; #1腔体机构单检步序号
ANDLD
LD=L(301) D1074 &0  ; #1腔体机构清氦步序号
OR=L(301) D1074 &1  ; #1腔体机构清氦步序号
ANDLD
LD=L(301) D1096 &0  ; #2腔体机构自动步序号
OR=L(301) D1096 &1  ; #2腔体机构自动步序号
ANDLD
LD=L(301) D1100 &0  ; #2腔体机构单检步序号
OR=L(301) D1100 &1  ; #2腔体机构单检步序号
ANDLD
LD=L(301) D1104 &0  ; #2腔体机构清氦步序号
OR=L(301) D1104 &1  ; #2腔体机构清氦步序号
ANDLD
LD=L(301) D1126 &0  ; #3腔体机构自动步序号
OR=L(301) D1126 &1  ; #3腔体机构自动步序号
ANDLD
LD=L(301) D1130 &0  ; #3腔体机构单检步序号
OR=L(301) D1130 &1  ; #3腔体机构单检步序号
ANDLD
LD=L(301) D1134 &0  ; #3腔体机构清氦步序号
OR=L(301) D1134 &1  ; #3腔体机构清氦步序号
ANDLD
LD=L(301) D1176 &0  ; #4腔体机构自动步序号
OR=L(301) D1176 &1  ; #4腔体机构自动步序号
ANDLD
LD=L(301) D1180 &0  ; #4腔体机构单检步序号
OR=L(301) D1180 &1  ; #4腔体机构单检步序号
ANDLD
LD=L(301) D1184 &0  ; #4腔体机构清氦步序号
OR=L(301) D1184 &1  ; #4腔体机构清氦步序号
ANDLD
OUT W3.00  ; 氦检单双检测选择允许

